P00021=-0.225,-6.128,-0.405,0.0000,0.0000,0.0000
P00022=0.222,-3.123,-1.508,0.0000,0.0000,0.0000
P00023=0.143,-0.036,0.682,0.0000,0.0000,0.0000
P00024=0.145,-0.552,1.326,0.0000,0.0000,0.0000
P00025=-2.003,0.006,0.728,0.0000,0.0000,0.0000
P00026=0.562,-0.002,-0.337,0.0000,0.0000,0.0000
P00027=-0.746,0.015,-9.096,0.0000,0.0000,0.0000
P00028=-2.237,-0.018,-7.702,0.0000,0.0000,0.0000
P00029=-2.156,-0.086,-4.681,0.0000,0.0000,0.0000
P00030=5.926,-4.294,-1.390,0.0000,0.0000,0.0000
P00031=1.853,-0.001,-1.549,0.0000,0.0000,0.0000
P00032=1.957,0.503,-7.217,0.0000,0.0000,0.0000
///RCONF 0,0,0,0,1,0,0,0,0,0,0,0,0,0,0,0,0,0,0,0,0,0,0,0
P00033=-0.123,0.612,-5.012,0.0000,0.0000,0.0000
///RCONF 0,0,0,0,0,0,0,0,0,0,0,0,0,0,0,0,0,0,0,0,0,0,0,0
P00034=-0.304,0.773,-2.693,0.0000,0.0000,0.0000
P00035=2.817,0.591,-1.622,0.0000,0.0000,0.0000
P00040=-0.030,9.648,2.467,0.0000,0.0000,0.0000
P00041=0.192,3.924,0.305,0.0000,0.0000,0.0000
P00042=-0.217,1.941,0.413,0.0000,0.0000,0.0000
P00043=-0.044,-1.937,1.197,0.0000,0.0000,0.0000
P00044=0.687,-2.322,1.156,0.0000,0.0000,0.0000
P00045=-0.068,-0.810,1.603,0.0000,0.0000,0.0000
P00046=0.799,0.043,1.292,0.0000,0.0000,0.0000
///RCONF 0,1,0,0,0,0,0,0,0,0,0,0,0,0,0,0,0,0,0,0,0,0,0,0
P00047=-0.011,1.737,-0.646,0.0000,0.0000,0.0000
///RCONF 0,0,0,0,0,0,0,0,0,0,0,0,0,0,0,0,0,0,0,0,0,0,0,0
P00048=2.411,0.025,-0.606,0.0000,0.0000,0.0000
P00049=3.413,-3.572,-1.618,0.0000,0.0000,0.0000
P00050=4.296,-4.501,-0.826,0.0000,0.0000,0.0000
P00051=0.367,3.892,0.009,0.0000,0.0000,0.0000
P00052=0.088,2.832,-0.342,0.0000,0.0000,0.0000
P00053=0.134,6.594,0.107,0.0000,0.0000,0.0000
P00054=-0.103,6.509,-0.702,0.0000,0.0000,0.0000
P00061=1.575,-3.405,-0.752,0.0000,0.0000,0.0000
P00062=-0.135,-0.848,-1.706,0.0000,0.0000,0.0000
P00063=0.036,-0.654,-3.005,0.0000,0.0000,0.0000
P00069=2.004,-0.013,0.498,0.0000,0.0000,0.0000
P00071=2.716,0.070,1.352,0.0000,0.0000,0.0000
P00072=1.041,-0.003,-0.797,0.0000,0.0000,0.0000
P00073=-0.961,5.319,-6.157,0.0000,0.0000,0.0000
P00074=1.123,1.944,-5.914,0.0000,0.0000,0.0000
P00080=-3.893,-3.240,-0.208,0.0000,0.0000,0.0000
P00081=19.486,11.347,1.262,0.0000,0.0000,0.0000
P00095=-3.945,4.918,-0.177,0.0000,0.0000,0.0000
P00096=-0.633,5.398,-3.809,0.0000,0.0000,0.0000
//INST
///DATE 2024/08/30 08:22
///ATTR SC,RW
///GROUP1 RB1,BS1
///GROUP2 ST1
NOP
'X2_8A-21A(90,0)
MOVJ C00000 BC00000 VJ=100.00  +MOVJ EC00000 VJ=100.00
CALL JOB:CLEAN-R1_KM_NEW
MOVJ C00001 BC00001 VJ=100.00  +MOVJ EC00001 VJ=100.00
MOVJ C00002 BC00002 VJ=100.00  +MOVJ EC00002 VJ=100.00
'Path S3463
SFTOF3D
MOVJ C00003 BC00003 VJ=100.00  +MOVJ EC00003 VJ=100.00
MOVL C00004 BC00004 V=666.7  +MOVJ EC00004 VJ=100.00
SMOVL C00005 BC00005 V=166.7  +MOVJ EC00005
SREFP 3 C00006 BC00006  +REFP EC00006
CALL JOB:SEARCH-R1-S13D
SET P095 P006
SFTON3D P095
SMOVL C00007 BC00007 V=166.7  +MOVJ EC00007
SMOVL C00008 BC00008 V=166.7  +MOVJ EC00008
SREFP 3 C00009 BC00009  +REFP EC00009
CALL JOB:SEARCH-R1-S13D
SET P095 P006
SFTON3D P095
SMOVL C00010 BC00010 V=166.7  +MOVJ EC00010
MOVL C00011 BC00011 V=1000.0  +MOVJ EC00011 VJ=100.00
'EndPath S3463
'Path S3464
SFTOF3D
MOVJ C00012 BC00012 VJ=100.00  +MOVJ EC00012 VJ=100.00
MOVL C00013 BC00013 V=666.7  +MOVJ EC00013 VJ=100.00
SMOVL C00014 BC00014 V=166.7  +MOVJ EC00014
SREFP 3 C00015 BC00015  +REFP EC00015
CALL JOB:SEARCH-R1-S13D
SET P096 P006
SFTON3D P096
SMOVL C00016 BC00016 V=166.7  +MOVJ EC00016
SREFP 3 C00017 BC00017  +REFP EC00017
CALL JOB:SEARCH-R1-S13D
SET P096 P006
SFTON3D P096
SMOVL C00018 BC00018 V=166.7  +MOVJ EC00018
MOVL C00019 BC00019 V=1000.0  +MOVJ EC00019 VJ=100.00
'EndPath S3464
'Path S3465
SFTOF3D
MOVJ C00020 BC00020 VJ=100.00  +MOVJ EC00020 VJ=100.00
MOVL C00021 BC00021 V=666.7  +MOVJ EC00021 VJ=100.00
SMOVL C00022 BC00022 V=166.7  +MOVJ EC00022
SREFP 3 C00023 BC00023  +REFP EC00023
CALL JOB:SEARCH-R1-S13D
SET P021 P006
SFTON3D P021
SMOVL C00024 BC00024 V=166.7  +MOVJ EC00024
SMOVL C00025 BC00025 V=166.7  +MOVJ EC00025
SREFP 3 C00026 BC00026  +REFP EC00026
CALL JOB:SEARCH-R1-S13D
SET P021 P006
SFTON3D P021
SMOVL C00027 BC00027 V=166.7  +MOVJ EC00027
MOVL C00028 BC00028 V=1000.0  +MOVJ EC00028 VJ=100.00
'EndPath S3465
'Path S3464
SFTOF3D
MOVJ C00029 BC00029 VJ=100.00  +MOVJ EC00029 VJ=100.00
MOVL C00030 BC00030 V=666.7  +MOVJ EC00030 VJ=100.00
SMOVL C00031 BC00031 V=166.7  +MOVJ EC00031
SREFP 3 C00032 BC00032  +REFP EC00032
CALL JOB:SEARCH-R1-S13D
SET P022 P006
SFTON3D P022
SMOVL C00033 BC00033 V=166.7  +MOVJ EC00033
SREFP 3 C00034 BC00034  +REFP EC00034
CALL JOB:SEARCH-R1-S13D
SET P022 P006
SFTON3D P022
SMOVL C00035 BC00035 V=166.7  +MOVJ EC00035
MOVL C00036 BC00036 V=1000.0  +MOVJ EC00036 VJ=100.00
'EndPath S3464
MOVJ C00037 BC00037 VJ=100.00  +MOVJ EC00037 VJ=100.00
'Path S3465
SFTOF3D
MOVJ C00038 BC00038 VJ=100.00  +MOVJ EC00038 VJ=100.00
MOVL C00039 BC00039 V=666.7  +MOVJ EC00039 VJ=100.00
SMOVL C00040 BC00040 V=166.7  +MOVJ EC00040
SREFP 3 C00041 BC00041  +REFP EC00041
CALL JOB:SEARCH-R1-S13D
SET P050 P006
SFTON3D P050
SMOVL C00042 BC00042 V=166.7  +MOVJ EC00042
SREFP 3 C00043 BC00043  +REFP EC00043
CALL JOB:SEARCH-R1-S13D
SET P050 P006
SFTON3D P050
SMOVL C00044 BC00044 V=166.7  +MOVJ EC00044
SMOVL C00045 BC00045 V=166.7  +MOVJ EC00045
SREFP 3 C00046 BC00046  +REFP EC00046
CALL JOB:SEARCH-R1-S13D
SET P050 P006
SFTON3D P050
SMOVL C00047 BC00047 V=166.7  +MOVJ EC00047
MOVL C00048 BC00048 V=1000.0  +MOVJ EC00048 VJ=100.00
'EndPath S3465
'Path S3466
SFTOF3D
MOVJ C00049 BC00049 VJ=100.00  +MOVJ EC00049 VJ=100.00
MOVL C00050 BC00050 V=666.7  +MOVJ EC00050 VJ=100.00
SMOVL C00051 BC00051 V=166.7  +MOVJ EC00051
SREFP 3 C00052 BC00052  +REFP EC00052
CALL JOB:SEARCH-R1-S13D
SET P051 P006
SFTON3D P051
SMOVL C00053 BC00053 V=166.7  +MOVJ EC00053
SREFP 3 C00054 BC00054  +REFP EC00054
CALL JOB:SEARCH-R1-S13D
SET P051 P006
SFTON3D P051
SMOVL C00055 BC00055 V=166.7  +MOVJ EC00055
SMOVL C00056 BC00056 V=250.0  +MOVJ EC00056
SREFP 3 C00057 BC00057  +REFP EC00057
CALL JOB:SEARCH-R1-S13D
SET P051 P006
SFTON3D P051
SMOVL C00058 BC00058 V=166.7  +MOVJ EC00058
MOVL C00059 BC00059 V=1000.0  +MOVJ EC00059 VJ=100.00
'EndPath S3466
MOVJ C00060 BC00060 VJ=100.00  +MOVJ EC00060 VJ=100.00
MOVJ C00061 BC00061 VJ=100.00  +MOVJ EC00061 VJ=100.00
'Path S3467
SFTOF3D
MOVJ C00062 BC00062 VJ=100.00  +MOVJ EC00062 VJ=100.00
MOVL C00063 BC00063 V=666.7  +MOVJ EC00063 VJ=100.00
SMOVL C00064 BC00064 V=166.7  +MOVJ EC00064
SREFP 3 C00065 BC00065  +REFP EC00065
CALL JOB:SEARCH-R1-S13D
SET P054 P006
SFTON3D P054
SMOVL C00066 BC00066 V=250.0  +MOVJ EC00066
SMOVL C00067 BC00067 V=166.7  +MOVJ EC00067
SREFP 3 C00068 BC00068  +REFP EC00068
CALL JOB:SEARCH-R1-S13D
SET P054 P006
SFTON3D P054
SMOVL C00069 BC00069 V=166.7  +MOVJ EC00069
SMOVL C00070 BC00070 V=800.0  +MOVJ EC00070
SMOVL C00071 BC00071 V=166.7  +MOVJ EC00071
SREFP 3 C00072 BC00072  +REFP EC00072
CALL JOB:SEARCH-R1-S13D
SET P054 P006
SFTON3D P054
SMOVL C00073 BC00073 V=166.7  +MOVJ EC00073
MOVL C00074 BC00074 V=1000.0  +MOVJ EC00074 VJ=100.00
'EndPath S3467
'Path S3475
SFTOF3D
MOVJ C00075 BC00075 VJ=100.00  +MOVJ EC00075 VJ=100.00
MOVL C00076 BC00076 V=666.7  +MOVJ EC00076 VJ=100.00
SMOVL C00077 BC00077 V=166.7  +MOVJ EC00077
SREFP 3 C00078 BC00078  +REFP EC00078
CALL JOB:SEARCH-R1-S13D
SET P034 P006
SFTON3D P034
SMOVL C00079 BC00079 V=166.7  +MOVJ EC00079
SMOVL C00080 BC00080 V=333.3  +MOVJ EC00080
SMOVL C00081 BC00081 V=166.7  +MOVJ EC00081
SREFP 3 C00082 BC00082  +REFP EC00082
CALL JOB:SEARCH-R1-S13D
SET P034 P006
SFTON3D P034
SMOVL C00083 BC00083 V=166.7  +MOVJ EC00083
SMOVL C00084 BC00084 V=166.7  +MOVJ EC00084
SREFP 3 C00085 BC00085  +REFP EC00085
CALL JOB:SEARCH-R1-S13D
SET P034 P006
SFTON3D P034
SMOVL C00086 BC00086 V=166.7  +MOVJ EC00086
MOVL C00087 BC00087 V=1000.0  +MOVJ EC00087 VJ=100.00
'EndPath S3475
'Path S3464
SFTOF3D
MOVJ C00088 BC00088 VJ=100.00  +MOVJ EC00088 VJ=100.00
MOVL C00089 BC00089 V=666.7  +MOVJ EC00089 VJ=100.00
SMOVL C00090 BC00090 V=166.7  +MOVJ EC00090
SREFP 3 C00091 BC00091  +REFP EC00091
CALL JOB:SEARCH-R1-S13D
SET P023 P006
SFTON3D P023
SMOVL C00092 BC00092 V=166.7  +MOVJ EC00092
SMOVL C00093 BC00093 V=500.0  +MOVJ EC00093
SMOVL C00094 BC00094 V=166.7  +MOVJ EC00094
SREFP 3 C00095 BC00095  +REFP EC00095
CALL JOB:SEARCH-R1-S13D
SET P023 P006
SFTON3D P023
SMOVL C00096 BC00096 V=166.7  +MOVJ EC00096
SMOVL C00097 BC00097 V=166.7  +MOVJ EC00097
SREFP 3 C00098 BC00098  +REFP EC00098
CALL JOB:SEARCH-R1-S13D
SET P023 P006
SFTON3D P023
SMOVL C00099 BC00099 V=166.7  +MOVJ EC00099
MOVL C00100 BC00100 V=1000.0  +MOVJ EC00100 VJ=100.00
MOVJ C00101 BC00101 VJ=80.00  +MOVJ EC00101 VJ=80.00
MOVJ C00102 BC00102 VJ=80.00  +MOVJ EC00102 VJ=80.00
SFTOF3D
MOVJ C00103 BC00103 VJ=80.00  +MOVJ EC00103 VJ=80.00
SMOVL C00104 BC00104 V=166.7  +MOVJ EC00104
SREFP 3 C00105 BC00105  +REFP EC00105
CALL JOB:SEARCH-R1-S13D
SET P061 P006
SFTON3D P061
SMOVL C00106 BC00106 V=166.7  +MOVJ EC00106
SREFP 3 C00107 BC00107  +REFP EC00107
CALL JOB:SEARCH-R1-S13D
SET P061 P006
SFTON3D P061
SMOVL C00108 BC00108 V=166.7  +MOVJ EC00108
SFTOF3D
SMOVL C00109 BC00109 V=500.0  +MOVJ EC00109
SMOVL C00110 BC00110 V=166.7  +MOVJ EC00110
SREFP 3 C00111 BC00111  +REFP EC00111
CALL JOB:SEARCH-R1-S13D
SET P062 P006
SFTON3D P062
SMOVL C00112 BC00112 V=166.7  +MOVJ EC00112
SREFP 3 C00113 BC00113  +REFP EC00113
CALL JOB:SEARCH-R1-S13D
SET P062 P006
SFTON3D P062
SMOVL C00114 BC00114 V=166.7  +MOVJ EC00114
SFTOF3D
SMOVL C00115 BC00115 V=500.0  +MOVJ EC00115
SMOVL C00116 BC00116 V=166.7  +MOVJ EC00116
SREFP 3 C00117 BC00117  +REFP EC00117
CALL JOB:SEARCH-R1-S13D
SET P063 P006
SFTON3D P063
SMOVL C00118 BC00118 V=166.7  +MOVJ EC00118
SREFP 3 C00119 BC00119  +REFP EC00119
CALL JOB:SEARCH-R1-S13D
SET P063 P006
SFTON3D P063
SMOVL C00120 BC00120 V=166.7  +MOVJ EC00120
SFTOF3D
SMOVL C00121 BC00121 V=500.0  +MOVJ EC00121
MOVJ C00122 BC00122 VJ=80.00  +MOVJ EC00122 VJ=80.00
MOVJ C00123 BC00123 VJ=80.00  +MOVJ EC00123 VJ=80.00
'EndPath S3464
MOVJ C00124 BC00124 VJ=100.00  +MOVJ EC00124 VJ=100.00
'Path S3465
SFTOF3D
MOVJ C00125 BC00125 VJ=100.00  +MOVJ EC00125 VJ=100.00
MOVL C00126 BC00126 V=666.7  +MOVJ EC00126 VJ=100.00
SMOVL C00127 BC00127 V=166.7  +MOVJ EC00127
SREFP 3 C00128 BC00128  +REFP EC00128
CALL JOB:SEARCH-R1-S13D
SET P024 P006
SFTON3D P024
SMOVL C00129 BC00129 V=166.7  +MOVJ EC00129
SREFP 3 C00130 BC00130  +REFP EC00130
CALL JOB:SEARCH-R1-S13D
SET P024 P006
SFTON3D P024
SMOVL C00131 BC00131 V=166.7  +MOVJ EC00131
SMOVL C00132 BC00132 V=166.7  +MOVJ EC00132
SREFP 3 C00133 BC00133  +REFP EC00133
CALL JOB:SEARCH-R1-S13D
SET P024 P006
SFTON3D P024
SMOVL C00134 BC00134 V=166.7  +MOVJ EC00134
MOVL C00135 BC00135 V=1000.0  +MOVJ EC00135 VJ=100.00
'EndPath S3465
'Path S3476
SFTOF3D
MOVJ C00136 BC00136 VJ=100.00  +MOVJ EC00136 VJ=100.00
MOVL C00137 BC00137 V=666.7  +MOVJ EC00137 VJ=100.00
SMOVL C00138 BC00138 V=166.7  +MOVJ EC00138
SREFP 3 C00139 BC00139  +REFP EC00139
CALL JOB:SEARCH-R1-S13D
SET P035 P006
SFTON3D P035
SMOVL C00140 BC00140 V=166.7  +MOVJ EC00140
SREFP 3 C00141 BC00141  +REFP EC00141
CALL JOB:SEARCH-R1-S13D
SET P035 P006
SFTON3D P035
SMOVL C00142 BC00142 V=166.7  +MOVJ EC00142
SMOVL C00143 BC00143 V=333.3  +MOVJ EC00143
SMOVL C00144 BC00144 V=166.7  +MOVJ EC00144
SREFP 3 C00145 BC00145  +REFP EC00145
CALL JOB:SEARCH-R1-S13D
SET P035 P006
SFTON3D P035
SMOVL C00146 BC00146 V=166.7  +MOVJ EC00146
MOVL C00147 BC00147 V=1000.0  +MOVJ EC00147 VJ=100.00
'EndPath S3476
'Path S3470
SFTOF3D
MOVJ C00148 BC00148 VJ=100.00  +MOVJ EC00148 VJ=100.00
MOVL C00149 BC00149 V=666.7  +MOVJ EC00149 VJ=100.00
SMOVL C00150 BC00150 V=166.7  +MOVJ EC00150
SREFP 3 C00151 BC00151  +REFP EC00151
CALL JOB:SEARCH-R1-S13D
SET P029 P006
SFTON3D P029
SMOVL C00152 BC00152 V=166.7  +MOVJ EC00152
SREFP 3 C00153 BC00153  +REFP EC00153
CALL JOB:SEARCH-R1-S13D
SET P029 P006
SFTON3D P029
SMOVL C00154 BC00154 V=166.7  +MOVJ EC00154
SMOVL C00155 BC00155 V=250.0  +MOVJ EC00155
SMOVL C00156 BC00156 V=166.7  +MOVJ EC00156
SREFP 3 C00157 BC00157  +REFP EC00157
CALL JOB:SEARCH-R1-S13D
SET P029 P006
SFTON3D P029
SMOVL C00158 BC00158 V=166.7  +MOVJ EC00158
MOVL C00159 BC00159 V=1000.0  +MOVJ EC00159 VJ=100.00
'EndPath S3470
'Path S4850
SFTOF3D
MOVL C00160 BC00160 V=666.7  +MOVJ EC00160 VJ=100.00
SMOVL C00161 BC00161 V=166.7  +MOVJ EC00161
SREFP 3 C00162 BC00162  +REFP EC00162
CALL JOB:SEARCH-R1-S13D
SET P071 P006
SFTON3D P071
SMOVL C00163 BC00163 V=166.7  +MOVJ EC00163
SREFP 3 C00164 BC00164  +REFP EC00164
CALL JOB:SEARCH-R1-S13D
SET P071 P006
SFTON3D P071
SMOVL C00165 BC00165 V=166.7  +MOVJ EC00165
SMOVL C00166 BC00166 V=166.7  +MOVJ EC00166
SREFP 3 C00167 BC00167  +REFP EC00167
CALL JOB:SEARCH-R1-S13D
SET P071 P006
SFTON3D P071
SMOVL C00168 BC00168 V=166.7  +MOVJ EC00168
MOVL C00169 BC00169 V=1000.0  +MOVJ EC00169 VJ=100.00
'EndPath S4850
'Path S4851
SFTOF3D
MOVJ C00170 BC00170 VJ=100.00  +MOVJ EC00170 VJ=100.00
'POMIAR_DOD_WZM_BOK
MOVL C00171 BC00171 V=666.7  +MOVJ EC00171 VJ=100.00
SMOVL C00172 BC00172 V=166.7  +MOVJ EC00172
SREFP 3 C00173 BC00173  +REFP EC00173
CALL JOB:SEARCH-R1-S13D
SET P080 P006
SFTON3D P080
SMOVL C00174 BC00174 V=166.7  +MOVJ EC00174
SREFP 3 C00175 BC00175  +REFP EC00175
CALL JOB:SEARCH-R1-S13D
SET P080 P006
SFTON3D P080
SMOVL C00176 BC00176 V=166.7  +MOVJ EC00176
SMOVL C00177 BC00177 V=250.0  +MOVJ EC00177
SMOVL C00178 BC00178 V=166.7  +MOVJ EC00178
SREFP 3 C00179 BC00179  +REFP EC00179
CALL JOB:SEARCH-R1-S13D
SET P080 P006
SFTON3D P080
SMOVL C00180 BC00180 V=166.7  +MOVJ EC00180
MOVL C00181 BC00181 V=1000.0  +MOVJ EC00181 VJ=100.00
SFTOF3D
MOVJ C00182 BC00182 VJ=100.00  +MOVJ EC00182 VJ=100.00
MOVL C00183 BC00183 V=666.7  +MOVJ EC00183 VJ=100.00
SMOVL C00184 BC00184 V=166.7  +MOVJ EC00184
SREFP 3 C00185 BC00185  +REFP EC00185
CALL JOB:SEARCH-R1-S13D
SET P072 P006
SFTON3D P072
SMOVL C00186 BC00186 V=166.7  +MOVJ EC00186
SREFP 3 C00187 BC00187  +REFP EC00187
CALL JOB:SEARCH-R1-S13D
SET P072 P006
SFTON3D P072
SMOVL C00188 BC00188 V=166.7  +MOVJ EC00188
MOVL C00189 BC00189 V=1000.0  +MOVJ EC00189 VJ=100.00
'EndPath S4851
MOVJ C00190 BC00190 VJ=100.00  +MOVJ EC00190 VJ=100.00
MOVJ C00191 BC00191 VJ=100.00  +MOVJ EC00191 VJ=100.00
'Path S4852
SFTOF3D
MOVJ C00192 BC00192 VJ=100.00  +MOVJ EC00192 VJ=100.00
MOVL C00193 BC00193 V=666.7  +MOVJ EC00193 VJ=100.00
SMOVL C00194 BC00194 V=166.7  +MOVJ EC00194
SREFP 3 C00195 BC00195  +REFP EC00195
CALL JOB:SEARCH-R1-S13D
SET P073 P006
SFTON3D P073
SMOVL C00196 BC00196 V=166.7  +MOVJ EC00196
SMOVL C00197 BC00197 V=166.7  +MOVJ EC00197
SREFP 3 C00198 BC00198  +REFP EC00198
CALL JOB:SEARCH-R1-S13D
SET P073 P006
SFTON3D P073
SMOVL C00199 BC00199 V=166.7  +MOVJ EC00199
SMOVL C00200 BC00200 V=166.7  +MOVJ EC00200
SREFP 3 C00201 BC00201  +REFP EC00201
CALL JOB:SEARCH-R1-S13D
SET P073 P006
SFTON3D P073
SMOVL C00202 BC00202 V=166.7  +MOVJ EC00202
MOVL C00203 BC00203 V=1000.0  +MOVJ EC00203 VJ=100.00
'EndPath S4852
MOVJ C00204 BC00204 VJ=100.00  +MOVJ EC00204 VJ=100.00
'Path S4853
SFTOF3D
MOVJ C00205 BC00205 VJ=100.00  +MOVJ EC00205 VJ=100.00
MOVL C00206 BC00206 V=666.7  +MOVJ EC00206 VJ=100.00
SMOVL C00207 BC00207 V=166.7  +MOVJ EC00207
SREFP 3 C00208 BC00208  +REFP EC00208
CALL JOB:SEARCH-R1-S13D
SET P074 P006
SFTON3D P074
SMOVL C00209 BC00209 V=166.7  +MOVJ EC00209
SREFP 3 C00210 BC00210  +REFP EC00210
CALL JOB:SEARCH-R1-S13D
SET P074 P006
SFTON3D P074
SMOVL C00211 BC00211 V=166.7  +MOVJ EC00211
MOVL C00212 BC00212 V=1000.0  +MOVJ EC00212 VJ=100.00
'EndPath S4853
'Path S3467
SFTOF3D
MOVJ C00213 BC00213 VJ=100.00  +MOVJ EC00213 VJ=100.00
MOVJ C00214 BC00214 VJ=100.00  +MOVJ EC00214 VJ=100.00
MOVL C00215 BC00215 V=666.7  +MOVJ EC00215 VJ=100.00
SMOVL C00216 BC00216 V=166.7  +MOVJ EC00216
SREFP 3 C00217 BC00217  +REFP EC00217
CALL JOB:SEARCH-R1-S13D
SET P081 P006
SFTON3D P081
SMOVL C00218 BC00218 V=166.7  +MOVJ EC00218
SMOVL C00219 BC00219 V=166.7  +MOVJ EC00219
SREFP 3 C00220 BC00220  +REFP EC00220
CALL JOB:SEARCH-R1-S13D
SET P081 P006
SFTON3D P081
SMOVL C00221 BC00221 V=166.7  +MOVJ EC00221
SMOVL C00222 BC00222 V=800.0  +MOVJ EC00222
SMOVL C00223 BC00223 V=166.7  +MOVJ EC00223
SREFP 3 C00224 BC00224  +REFP EC00224
CALL JOB:SEARCH-R1-S13D
SET P081 P006
SFTON3D P081
SMOVL C00225 BC00225 V=166.7  +MOVJ EC00225
MOVJ C00226 BC00226 VJ=100.00  +MOVJ EC00226 VJ=100.00
MOVJ C00227 BC00227 VJ=100.00  +MOVJ EC00227 VJ=100.00
SFTOF3D
MOVJ C00228 BC00228 VJ=100.00  +MOVJ EC00228 VJ=100.00
MOVL C00229 BC00229 V=666.7  +MOVJ EC00229 VJ=100.00
SMOVL C00230 BC00230 V=166.7  +MOVJ EC00230
SREFP 3 C00231 BC00231  +REFP EC00231
CALL JOB:SEARCH-R1-S13D
SET P026 P006
SFTON3D P026
SMOVL C00232 BC00232 V=166.7  +MOVJ EC00232
SREFP 3 C00233 BC00233  +REFP EC00233
CALL JOB:SEARCH-R1-S13D
SET P026 P006
SFTON3D P026
SMOVL C00234 BC00234 V=166.7  +MOVJ EC00234
SMOVL C00235 BC00235 V=800.0  +MOVJ EC00235
SMOVL C00236 BC00236 V=166.7  +MOVJ EC00236
SREFP 3 C00237 BC00237  +REFP EC00237
CALL JOB:SEARCH-R1-S13D
SET P026 P006
SFTON3D P026
SMOVL C00238 BC00238 V=166.7  +MOVJ EC00238
MOVL C00239 BC00239 V=1000.0  +MOVJ EC00239 VJ=100.00
'EndPath S3467
MOVJ C00240 BC00240 VJ=100.00  +MOVJ EC00240 VJ=100.00
'Path S3466
SFTOF3D
MOVJ C00241 BC00241 VJ=100.00  +MOVJ EC00241 VJ=100.00
MOVL C00242 BC00242 V=666.7  +MOVJ EC00242 VJ=100.00
SMOVL C00243 BC00243 V=166.7  +MOVJ EC00243
SREFP 3 C00244 BC00244  +REFP EC00244
CALL JOB:SEARCH-R1-S13D
SET P025 P006
SFTON3D P025
SMOVL C00245 BC00245 V=166.7  +MOVJ EC00245
SMOVL C00246 BC00246 V=166.7  +MOVJ EC00246
SREFP 3 C00247 BC00247  +REFP EC00247
CALL JOB:SEARCH-R1-S13D
SET P025 P006
SFTON3D P025
SMOVL C00248 BC00248 V=166.7  +MOVJ EC00248
SMOVL C00249 BC00249 V=200.0  +MOVJ EC00249
SMOVL C00250 BC00250 V=166.7  +MOVJ EC00250
SREFP 3 C00251 BC00251  +REFP EC00251
CALL JOB:SEARCH-R1-S13D
SET P025 P006
SFTON3D P025
SMOVL C00252 BC00252 V=166.7  +MOVJ EC00252
MOVL C00253 BC00253 V=1000.0  +MOVJ EC00253 VJ=100.00
'EndPath S3466
MOVJ C00254 BC00254 VJ=100.00  +MOVJ EC00254 VJ=100.00
'Path S3469
SFTOF3D
MOVJ C00255 BC00255 VJ=100.00  +MOVJ EC00255 VJ=100.00
MOVL C00256 BC00256 V=666.7  +MOVJ EC00256 VJ=100.00
SMOVL C00257 BC00257 V=166.7  +MOVJ EC00257
SREFP 3 C00258 BC00258  +REFP EC00258
CALL JOB:SEARCH-R1-S13D
SET P028 P006
SFTON3D P028
SMOVL C00259 BC00259 V=166.7  +MOVJ EC00259
SREFP 3 C00260 BC00260  +REFP EC00260
CALL JOB:SEARCH-R1-S13D
SET P028 P006
SFTON3D P028
SMOVL C00261 BC00261 V=166.7  +MOVJ EC00261
SMOVL C00262 BC00262 V=333.3  +MOVJ EC00262
SMOVL C00263 BC00263 V=166.7  +MOVJ EC00263
SREFP 3 C00264 BC00264  +REFP EC00264
CALL JOB:SEARCH-R1-S13D
SET P028 P006
SFTON3D P028
SMOVL C00265 BC00265 V=166.7  +MOVJ EC00265
MOVL C00266 BC00266 V=1000.0  +MOVJ EC00266 VJ=100.00
'EndPath S3469
MOVJ C00267 BC00267 VJ=100.00  +MOVJ EC00267 VJ=100.00
'Path S3474
SFTOF3D
MOVJ C00268 BC00268 VJ=100.00  +MOVJ EC00268 VJ=100.00
MOVL C00269 BC00269 V=666.7  +MOVJ EC00269 VJ=100.00
SMOVL C00270 BC00270 V=166.7  +MOVJ EC00270
SREFP 3 C00271 BC00271  +REFP EC00271
CALL JOB:SEARCH-R1-S13D
SET P033 P006
SFTON3D P033
SMOVL C00272 BC00272 V=166.7  +MOVJ EC00272
SREFP 3 C00273 BC00273  +REFP EC00273
CALL JOB:SEARCH-R1-S13D
SET P033 P006
SFTON3D P033
SMOVL C00274 BC00274 V=166.7  +MOVJ EC00274
SMOVL C00275 BC00275 V=250.0  +MOVJ EC00275
SMOVL C00276 BC00276 V=166.7  +MOVJ EC00276
SREFP 3 C00277 BC00277  +REFP EC00277
CALL JOB:SEARCH-R1-S13D
SET P033 P006
SFTON3D P033
SMOVL C00278 BC00278 V=166.7  +MOVJ EC00278
MOVL C00279 BC00279 V=1000.0  +MOVJ EC00279 VJ=100.00
'EndPath S3474
'Path S3468
SFTOF3D
MOVJ C00280 BC00280 VJ=100.00  +MOVJ EC00280 VJ=100.00
MOVL C00281 BC00281 V=666.7  +MOVJ EC00281 VJ=100.00
SMOVL C00282 BC00282 V=166.7  +MOVJ EC00282
SREFP 3 C00283 BC00283  +REFP EC00283
CALL JOB:SEARCH-R1-S13D
SET P027 P006
SFTON3D P027
SMOVL C00284 BC00284 V=166.7  +MOVJ EC00284
SMOVL C00285 BC00285 V=166.7  +MOVJ EC00285
SREFP 3 C00286 BC00286  +REFP EC00286
CALL JOB:SEARCH-R1-S13D
SET P027 P006
SFTON3D P027
SMOVL C00287 BC00287 V=166.7  +MOVJ EC00287
SMOVL C00288 BC00288 V=166.7  +MOVJ EC00288
SREFP 3 C00289 BC00289  +REFP EC00289
CALL JOB:SEARCH-R1-S13D
SET P027 P006
SFTON3D P027
SMOVL C00290 BC00290 V=166.7  +MOVJ EC00290
MOVL C00291 BC00291 V=1000.0  +MOVJ EC00291 VJ=100.00
'EndPath S3468
'Path S3471
SFTOF3D
MOVJ C00292 BC00292 VJ=100.00  +MOVJ EC00292 VJ=100.00
MOVL C00293 BC00293 V=666.7  +MOVJ EC00293 VJ=100.00
SMOVL C00294 BC00294 V=166.7  +MOVJ EC00294
SREFP 3 C00295 BC00295  +REFP EC00295
CALL JOB:SEARCH-R1-S13D
SET P030 P006
SFTON3D P030
SMOVL C00296 BC00296 V=166.7  +MOVJ EC00296
SREFP 3 C00297 BC00297  +REFP EC00297
CALL JOB:SEARCH-R1-S13D
SET P030 P006
SFTON3D P030
SMOVL C00298 BC00298 V=166.7  +MOVJ EC00298
MOVL C00299 BC00299 V=1000.0  +MOVJ EC00299 VJ=100.00
'EndPath S3471
'Path S3472
SFTOF3D
MOVJ C00300 BC00300 VJ=100.00  +MOVJ EC00300 VJ=100.00
MOVL C00301 BC00301 V=666.7  +MOVJ EC00301 VJ=100.00
SMOVL C00302 BC00302 V=166.7  +MOVJ EC00302
SREFP 3 C00303 BC00303  +REFP EC00303
CALL JOB:SEARCH-R1-S13D
SET P031 P006
SFTON3D P031
SMOVL C00304 BC00304 V=166.7  +MOVJ EC00304
SREFP 3 C00305 BC00305  +REFP EC00305
CALL JOB:SEARCH-R1-S13D
SET P031 P006
SFTON3D P031
SMOVL C00306 BC00306 V=166.7  +MOVJ EC00306
MOVL C00307 BC00307 V=1000.0  +MOVJ EC00307 VJ=100.00
'EndPath S3472
MOVJ C00308 BC00308 VJ=100.00  +MOVJ EC00308 VJ=100.00
'Path S3472
SFTOF3D
MOVJ C00309 BC00309 VJ=100.00  +MOVJ EC00309 VJ=100.00
MOVL C00310 BC00310 V=666.7  +MOVJ EC00310 VJ=100.00
SMOVL C00311 BC00311 V=166.7  +MOVJ EC00311
SREFP 3 C00312 BC00312  +REFP EC00312
CALL JOB:SEARCH-R1-S13D
SET P032 P006
SFTON3D P032
SMOVL C00313 BC00313 V=166.7  +MOVJ EC00313
SREFP 3 C00314 BC00314  +REFP EC00314
CALL JOB:SEARCH-R1-S13D
SET P032 P006
SFTON3D P032
SMOVL C00315 BC00315 V=166.7  +MOVJ EC00315
SMOVL C00316 BC00316 V=133.3  +MOVJ EC00316
SREFP 3 C00317 BC00317  +REFP EC00317
CALL JOB:SEARCH-R1-S13D
SET P032 P006
SFTON3D P032
SMOVL C00318 BC00318 V=166.7  +MOVJ EC00318
MOVL C00319 BC00319 V=1000.0  +MOVJ EC00319 VJ=100.00
'EndPath S3472
MOVJ C00320 BC00320 VJ=100.00  +MOVJ EC00320 VJ=100.00
'Path S3477
SFTOF3D
MOVJ C00321 BC00321 VJ=100.00  +MOVJ EC00321 VJ=100.00
SMOVL C00322 BC00322 V=166.7  +MOVJ EC00322
SREFP 3 C00323 BC00323  +REFP EC00323
CALL JOB:SEARCH-R1-S13D
SET P069 P006
SFTON3D P069
SMOVL C00324 BC00324 V=250.0  +MOVJ EC00324
SMOVL C00325 BC00325 V=250.0  +MOVJ EC00325
SMOVL C00326 BC00326 V=166.7  +MOVJ EC00326
SREFP 3 C00327 BC00327  +REFP EC00327
CALL JOB:SEARCH-R1-S13D
SET P069 P006
SFTON3D P069
SMOVL C00328 BC00328 V=166.7  +MOVJ EC00328
SFTOF3D
SMOVL C00329 BC00329 V=666.7  +MOVJ EC00329
MOVL C00330 BC00330 V=666.7  +MOVJ EC00330 VJ=100.00
SMOVL C00331 BC00331 V=166.7  +MOVJ EC00331
SREFP 3 C00332 BC00332  +REFP EC00332
CALL JOB:SEARCH-R1-S13D
SET P052 P006
SFTON3D P052
SMOVL C00333 BC00333 V=166.7  +MOVJ EC00333
SREFP 3 C00334 BC00334  +REFP EC00334
CALL JOB:SEARCH-R1-S13D
SET P052 P006
SFTON3D P052
SMOVL C00335 BC00335 V=166.7  +MOVJ EC00335
MOVL C00336 BC00336 V=1000.0  +MOVJ EC00336 VJ=100.00
'EndPath S3477
MOVJ C00337 BC00337 VJ=100.00  +MOVJ EC00337 VJ=100.00
'poprawiÄ searcha- nie mialem
'wyciecia
'Path S3478
SFTOF3D
MOVJ C00338 BC00338 VJ=100.00  +MOVJ EC00338 VJ=100.00
MOVL C00339 BC00339 V=666.7  +MOVJ EC00339 VJ=100.00
SMOVL C00340 BC00340 V=166.7  +MOVJ EC00340
SREFP 3 C00341 BC00341  +REFP EC00341
CALL JOB:SEARCH-R1-S13D
SET P053 P006
SFTON3D P053
SMOVL C00342 BC00342 V=166.7  +MOVJ EC00342
SREFP 3 C00343 BC00343  +REFP EC00343
CALL JOB:SEARCH-R1-S13D
SET P053 P006
SFTON3D P053
SMOVL C00344 BC00344 V=166.7  +MOVJ EC00344
MOVL C00345 BC00345 V=1000.0  +MOVJ EC00345 VJ=100.00
'EndPath S3478
'
MOVJ C00346 BC00346 VJ=100.00  +MOVJ EC00346 VJ=100.00
'Path W3476
SFTOF3D
SFTON3D P033
MOVJ C00347 BC00347 VJ=100.00  +MOVJ EC00347 VJ=100.00
SMOVL C00348 BC00348 V=800.0  +MOVJ EC00348
SMOVL C00349 BC00349 V=166.7 PL=0  +MOVJ EC00349
MACRO1 MJ#(0) ARGF14
ARCON
SMOVL C00350 BC00350 V=10.0  +MOVJ EC00350
ARCOF
SMOVL C00351 BC00351 V=800.0  +MOVJ EC00351
SMOVL C00352 BC00352 V=1000.0  +MOVJ EC00352
SFTOF3D
'EndPath W3476
'Path W3477
SFTOF3D
SFTON3D P033
MOVJ C00353 BC00353 VJ=100.00  +MOVJ EC00353 VJ=100.00
SMOVL C00354 BC00354 V=800.0  +MOVJ EC00354
SMOVL C00355 BC00355 V=166.7 PL=0  +MOVJ EC00355
SMOVL C00356 BC00356 V=10.0  +MOVJ EC00356
SMOVL C00357 BC00357 V=10.0  +MOVJ EC00357
SMOVL C00358 BC00358 V=10.0  +MOVJ EC00358
ARCOF
SMOVL C00359 BC00359 V=800.0  +MOVJ EC00359
SMOVL C00360 BC00360 V=1000.0  +MOVJ EC00360
SFTOF3D
'EndPath W3477
MOVJ C00361 BC00361 VJ=100.00  +MOVJ EC00361 VJ=100.00
'Path W3478
SFTOF3D
SFTON3D P033
MOVJ C00362 BC00362 VJ=100.00  +MOVJ EC00362 VJ=100.00
SMOVL C00363 BC00363 V=800.0  +MOVJ EC00363
SMOVL C00364 BC00364 V=166.7 PL=0  +MOVJ EC00364
ARCON
SMOVL C00365 BC00365 V=10.0  +MOVJ EC00365
SMOVL C00366 BC00366 V=10.0  +MOVJ EC00366
SMOVL C00367 BC00367 V=10.0  +MOVJ EC00367
ARCOF
SMOVL C00368 BC00368 V=800.0  +MOVJ EC00368
SMOVL C00369 BC00369 V=1000.0  +MOVJ EC00369
SFTOF3D
'EndPath W3478
MOVJ C00370 BC00370 VJ=100.00  +MOVJ EC00370 VJ=100.00
MOVJ C00371 BC00371 VJ=100.00  +MOVJ EC00371 VJ=100.00
SFTOF3D
SFTON3D P081
MOVJ C00372 BC00372 VJ=100.00  +MOVJ EC00372 VJ=100.00
SMOVL C00373 BC00373 V=800.0  +MOVJ EC00373
SMOVL C00374 BC00374 V=166.7 PL=0  +MOVJ EC00374
ARCON
SMOVL C00375 BC00375 V=9.2  +MOVJ EC00375
ARCOF
SMOVL C00376 BC00376 V=800.0  +MOVJ EC00376
SMOVL C00377 BC00377 V=1000.0  +MOVJ EC00377
SFTOF3D
'EndPath W3479
'Path W3480
SFTOF3D
SFTON3D P081
MOVJ C00378 BC00378 VJ=100.00  +MOVJ EC00378 VJ=100.00
SMOVL C00379 BC00379 V=800.0  +MOVJ EC00379
SMOVL C00380 BC00380 V=150.0 PL=0  +MOVJ EC00380
ARCON
SMOVL C00381 BC00381 V=10.0  +MOVJ EC00381
ARCOF
SMOVL C00382 BC00382 V=800.0  +MOVJ EC00382
SMOVL C00383 BC00383 V=1000.0  +MOVJ EC00383
SFTOF3D
'EndPath W3480
'Path W3481
SFTOF3D
SFTON3D P081
MOVJ C00384 BC00384 VJ=100.00  +MOVJ EC00384 VJ=100.00
SMOVL C00385 BC00385 V=800.0  +MOVJ EC00385
SMOVL C00386 BC00386 V=150.0 PL=0  +MOVJ EC00386
ARCON
SMOVL C00387 BC00387 V=10.0  +MOVJ EC00387
ARCOF
SMOVL C00388 BC00388 V=800.0  +MOVJ EC00388
SMOVL C00389 BC00389 V=1000.0  +MOVJ EC00389
SFTOF3D
'EndPath W3481
MOVJ C00390 BC00390 VJ=100.00  +MOVJ EC00390 VJ=100.00
'uwaga na podajnik
'Path W3481
SFTOF3D
SFTON3D P081
MOVJ C00391 BC00391 VJ=50.00  +MOVJ EC00391 VJ=15.00
SMOVL C00392 BC00392 V=800.0  +MOVJ EC00392
SMOVL C00393 BC00393 V=150.0 PL=0  +MOVJ EC00393
ARCON
SMOVL C00394 BC00394 V=10.0  +MOVJ EC00394
ARCOF
SMOVL C00395 BC00395 V=800.0  +MOVJ EC00395
SMOVL C00396 BC00396 V=1000.0  +MOVJ EC00396
SFTOF3D
'9
'Path W3479
MOVJ C00397 BC00397 VJ=100.00  +MOVJ EC00397 VJ=100.00
SFTOF3D
SFTON3D P026
MOVJ C00398 BC00398 VJ=100.00  +MOVJ EC00398 VJ=100.00
SMOVL C00399 BC00399 V=800.0  +MOVJ EC00399
SMOVL C00400 BC00400 V=166.7 PL=0  +MOVJ EC00400
ARCON
SMOVL C00401 BC00401 V=9.2  +MOVJ EC00401
SMOVL C00402 BC00402 V=9.2  +MOVJ EC00402
SMOVL C00403 BC00403 V=9.2  +MOVJ EC00403
ARCOF
SMOVL C00404 BC00404 V=800.0  +MOVJ EC00404
SMOVL C00405 BC00405 V=1000.0  +MOVJ EC00405
SFTOF3D
'EndPath W3479
'Path W3480
SFTOF3D
SFTON3D P026
MOVJ C00406 BC00406 VJ=100.00  +MOVJ EC00406 VJ=100.00
SMOVL C00407 BC00407 V=800.0  +MOVJ EC00407
SMOVL C00408 BC00408 V=150.0 PL=0  +MOVJ EC00408
ARCON
SMOVL C00409 BC00409 V=10.0  +MOVJ EC00409
SMOVL C00410 BC00410 V=10.0  +MOVJ EC00410
SMOVL C00411 BC00411 V=10.0  +MOVJ EC00411
ARCOF
SMOVL C00412 BC00412 V=800.0  +MOVJ EC00412
SMOVL C00413 BC00413 V=1000.0  +MOVJ EC00413
SFTOF3D
'EndPath W3480
'Path W3481
SFTOF3D
SFTON3D P026
MOVJ C00414 BC00414 VJ=100.00  +MOVJ EC00414 VJ=100.00
SMOVL C00415 BC00415 V=800.0  +MOVJ EC00415
SMOVL C00416 BC00416 V=150.0 PL=0  +MOVJ EC00416
ARCON
SMOVL C00417 BC00417 V=10.0  +MOVJ EC00417
ARCOF
SMOVL C00418 BC00418 V=800.0  +MOVJ EC00418
SMOVL C00419 BC00419 V=1000.0  +MOVJ EC00419
SFTOF3D
'EndPath W3481
MOVJ C00420 BC00420 VJ=100.00  +MOVJ EC00420 VJ=100.00
'uwaga na podajnik
'Path W3481
SFTOF3D
SFTON3D P026
MOVJ C00421 BC00421 VJ=50.00  +MOVJ EC00421 VJ=15.00
SMOVL C00422 BC00422 V=800.0  +MOVJ EC00422
SMOVL C00423 BC00423 V=150.0 PL=0  +MOVJ EC00423
ARCON
SMOVL C00424 BC00424 V=10.0  +MOVJ EC00424
SMOVL C00425 BC00425 V=10.0  +MOVJ EC00425
ARCOF
SMOVL C00426 BC00426 V=800.0  +MOVJ EC00426
SMOVL C00427 BC00427 V=1000.0  +MOVJ EC00427
SFTOF3D
'EndPath W3481
'brak dostepu offset drutu 1cm
'Path W3482
SFTOF3D
SFTON3D P026
MOVJ C00428 BC00428 VJ=100.00  +MOVJ EC00428 VJ=100.00
SMOVL C00429 BC00429 V=800.0  +MOVJ EC00429
SMOVL C00430 BC00430 V=150.0 PL=0  +MOVJ EC00430
ARCON
SMOVL C00431 BC00431 V=10.0  +MOVJ EC00431
ARCOF
SMOVL C00432 BC00432 V=800.0  +MOVJ EC00432
SMOVL C00433 BC00433 V=1000.0  +MOVJ EC00433
SFTOF3D
'EndPath W3482
MOVJ C00434 BC00434 VJ=100.00  +MOVJ EC00434 VJ=100.00
MOVJ C00435 BC00435 VJ=100.00  +MOVJ EC00435 VJ=100.00
'10
'11
'Path W3484
SFTOF3D
SFTON3D P025
MOVJ C00436 BC00436 VJ=100.00  +MOVJ EC00436 VJ=100.00
SMOVL C00437 BC00437 V=800.0  +MOVJ EC00437
SMOVL C00438 BC00438 V=150.0 PL=0  +MOVJ EC00438
ARCON
SMOVL C00439 BC00439 V=10.0  +MOVJ EC00439
SMOVL C00440 BC00440 V=10.0  +MOVJ EC00440
ARCOF
SMOVL C00441 BC00441 V=800.0  +MOVJ EC00441
SMOVL C00442 BC00442 V=1000.0  +MOVJ EC00442
SFTOF3D
'EndPath W3484
MOVJ C00443 BC00443 VJ=100.00  +MOVJ EC00443 VJ=100.00
'brak dostepu offset drutu 1cm
'Path W3483
SFTOF3D
SFTON3D P025
MOVJ C00444 BC00444 VJ=100.00  +MOVJ EC00444 VJ=100.00
SMOVL C00445 BC00445 V=800.0  +MOVJ EC00445
SMOVL C00446 BC00446 V=166.7 PL=0  +MOVJ EC00446
ARCON
SMOVL C00447 BC00447 V=10.0  +MOVJ EC00447
ARCOF
SMOVL C00448 BC00448 V=800.0  +MOVJ EC00448
SMOVL C00449 BC00449 V=1000.0  +MOVJ EC00449
SFTOF3D
'EndPath W3483
MOVJ C00450 BC00450 VJ=100.00  +MOVJ EC00450 VJ=100.00
MOVJ C00451 BC00451 VJ=100.00  +MOVJ EC00451 VJ=100.00
MOVJ C00452 BC00452 VJ=100.00  +MOVJ EC00452 VJ=100.00
'Path W4854
SFTOF3D
SFTON3D P073
MOVJ C00453 BC00453 VJ=100.00  +MOVJ EC00453 VJ=100.00
SMOVL C00454 BC00454 V=800.0  +MOVJ EC00454
SMOVL C00455 BC00455 V=150.0 PL=0  +MOVJ EC00455
MACRO1 MJ#(0) ARGF9
ARCON
SMOVL C00456 BC00456 V=9.2  +MOVJ EC00456
SFTON3D P074
SMOVL C00457 BC00457 V=9.2  +MOVJ EC00457
SMOVL C00458 BC00458 V=9.2  +MOVJ EC00458
ARCOF
SMOVL C00459 BC00459 V=800.0  +MOVJ EC00459
MOVJ C00460 BC00460 VJ=50.00  +MOVJ EC00460 VJ=100.00
SMOVL C00461 BC00461 V=166.7  +MOVJ EC00461
SMOVL C00462 BC00462 V=166.7  +MOVJ EC00462
SMOVL C00463 BC00463 V=50.0 PL=0  +MOVJ EC00463
ARCON
SMOVL C00464 BC00464 V=9.2  +MOVJ EC00464
SMOVL C00465 BC00465 V=9.2  +MOVJ EC00465
ARCOF
SMOVL C00466 BC00466 V=1000.0  +MOVJ EC00466
SFTOF3D
'EndPath W4854
'12
MOVJ C00467 BC00467 VJ=100.00  +MOVJ EC00467 VJ=100.00
MOVJ C00468 BC00468 VJ=100.00  +MOVJ EC00468 VJ=100.00
MOVJ C00469 BC00469 VJ=100.00  +MOVJ EC00469 VJ=100.00
'Path W3485
SFTOF3D
SFTON3D P034
MOVJ C00470 BC00470 VJ=100.00  +MOVJ EC00470 VJ=100.00
SMOVL C00471 BC00471 V=800.0  +MOVJ EC00471
SMOVL C00472 BC00472 V=150.0 PL=0  +MOVJ EC00472
MACRO1 MJ#(0) ARGF14
ARCON
SMOVL C00473 BC00473 V=10.0  +MOVJ EC00473
SMOVL C00474 BC00474 V=10.0  +MOVJ EC00474
SMOVL C00475 BC00475 V=10.0  +MOVJ EC00475
ARCOF
SMOVL C00476 BC00476 V=800.0  +MOVJ EC00476
SMOVL C00477 BC00477 V=1000.0  +MOVJ EC00477
SFTOF3D
MOVJ C00478 BC00478 VJ=80.00  +MOVJ EC00478 VJ=80.00
MOVJ C00479 BC00479 VJ=80.00  +MOVJ EC00479 VJ=80.00
MOVJ C00480 BC00480 VJ=80.00  +MOVJ EC00480 VJ=80.00
MACRO1 MJ#(0) ARGF6
SFTON3D P063
SMOVL C00481 BC00481 V=166.7  +MOVJ EC00481
ARCON
SMOVL C00482 BC00482 V=11.7  +MOVJ EC00482
SMOVL C00483 BC00483 V=11.7  +MOVJ EC00483
SFTON3D P062
SMOVL C00484 BC00484 V=11.0  +MOVJ EC00484
SMOVL C00485 BC00485 V=11.0  +MOVJ EC00485
SFTON3D P061
SMOVL C00486 BC00486 V=11.0  +MOVJ EC00486
SMOVL C00487 BC00487 V=11.0  +MOVJ EC00487
ARCOF
SMOVL C00488 BC00488 V=800.0  +MOVJ EC00488
SFTOF3D
MOVJ C00489 BC00489 VJ=80.00  +MOVJ EC00489 VJ=80.00
MOVJ C00490 BC00490 VJ=80.00  +MOVJ EC00490 VJ=80.00
MOVJ C00491 BC00491 VJ=80.00  +MOVJ EC00491 VJ=80.00
'EndPath W3485
'Path W3486
SFTOF3D
SFTON3D P050
MOVJ C00492 BC00492 VJ=100.00  +MOVJ EC00492 VJ=100.00
SMOVL C00493 BC00493 V=800.0  +MOVJ EC00493
SMOVL C00494 BC00494 V=150.0 PL=0  +MOVJ EC00494
MACRO1 MJ#(0) ARGF14
ARCON
SMOVL C00495 BC00495 V=10.0  +MOVJ EC00495
SMOVL C00496 BC00496 V=10.0  +MOVJ EC00496
SMOVL C00497 BC00497 V=10.0  +MOVJ EC00497
ARCOF
SMOVL C00498 BC00498 V=800.0  +MOVJ EC00498
SMOVL C00499 BC00499 V=1000.0  +MOVJ EC00499
SFTOF3D
'EndPath W3486
MOVJ C00500 BC00500 VJ=100.00  +MOVJ EC00500 VJ=100.00
'Path W3485
SFTOF3D
SFTON3D P034
MOVJ C00501 BC00501 VJ=100.00  +MOVJ EC00501 VJ=100.00
SMOVL C00502 BC00502 V=800.0  +MOVJ EC00502
SMOVL C00503 BC00503 V=166.7 PL=0  +MOVJ EC00503
ARCON
SMOVL C00504 BC00504 V=9.2  +MOVJ EC00504
SMOVL C00505 BC00505 V=9.2  +MOVJ EC00505
SMOVL C00506 BC00506 V=9.2  +MOVJ EC00506
ARCOF
SMOVL C00507 BC00507 V=800.0  +MOVJ EC00507
SMOVL C00508 BC00508 V=1000.0  +MOVJ EC00508
SFTOF3D
'EndPath W3485
'Path W3487
SFTOF3D
SFTON3D P054
MOVJ C00509 BC00509 VJ=100.00  +MOVJ EC00509 VJ=100.00
SMOVL C00510 BC00510 V=800.0  +MOVJ EC00510
SMOVL C00511 BC00511 V=150.0 PL=0  +MOVJ EC00511
ARCON
SMOVL C00512 BC00512 V=9.2  +MOVJ EC00512
SMOVL C00513 BC00513 V=9.2  +MOVJ EC00513
SMOVL C00514 BC00514 V=9.2  +MOVJ EC00514
ARCOF
SMOVL C00515 BC00515 V=800.0  +MOVJ EC00515
SMOVL C00516 BC00516 V=1000.0  +MOVJ EC00516
SFTOF3D
'EndPath W3487
MOVJ C00517 BC00517 VJ=100.00  +MOVJ EC00517 VJ=100.00
'Path W3487
SFTOF3D
SFTON3D P028
MOVJ C00518 BC00518 VJ=100.00  +MOVJ EC00518 VJ=100.00
SMOVL C00519 BC00519 V=800.0  +MOVJ EC00519
SMOVL C00520 BC00520 V=150.0 PL=0  +MOVJ EC00520
ARCON
SMOVL C00521 BC00521 V=9.2  +MOVJ EC00521
SMOVL C00522 BC00522 V=9.2  +MOVJ EC00522
SMOVL C00523 BC00523 V=9.2  +MOVJ EC00523
ARCOF
SMOVL C00524 BC00524 V=800.0  +MOVJ EC00524
SMOVL C00525 BC00525 V=1000.0  +MOVJ EC00525
SFTOF3D
'EndPath W3487
MOVJ C00526 BC00526 VJ=100.00  +MOVJ EC00526 VJ=100.00
MOVJ C00527 BC00527 VJ=100.00  +MOVJ EC00527 VJ=100.00
'brak dostepu offset 5mm
'Path W3488
SFTOF3D
SFTON3D P028
MOVJ C00528 BC00528 VJ=100.00  +MOVJ EC00528 VJ=100.00
SMOVL C00529 BC00529 V=800.0  +MOVJ EC00529
SMOVL C00530 BC00530 V=150.0 PL=0  +MOVJ EC00530
ARCON
SMOVL C00531 BC00531 V=11.7  +MOVJ EC00531
ARCOF
SMOVL C00532 BC00532 V=800.0  +MOVJ EC00532
SMOVL C00533 BC00533 V=1000.0  +MOVJ EC00533
SFTOF3D
'EndPath W3488
MOVJ C00534 BC00534 VJ=100.00  +MOVJ EC00534 VJ=100.00
'13
'Path W3489
SFTOF3D
SFTON3D P030
MOVJ C00535 BC00535 VJ=100.00  +MOVJ EC00535 VJ=100.00
SMOVL C00536 BC00536 V=800.0  +MOVJ EC00536
SMOVL C00537 BC00537 V=150.0 PL=0  +MOVJ EC00537
MACRO1 MJ#(0) ARGF9
ARCON
SFTON3D P031
SMOVL C00538 BC00538 V=10.8  +MOVJ EC00538
ARCOF
SMOVL C00539 BC00539 V=800.0  +MOVJ EC00539
SMOVL C00540 BC00540 V=1000.0  +MOVJ EC00540
SFTOF3D
'EndPath W3489
'Path W3490
SFTOF3D
MOVJ C00541 BC00541 VJ=100.00  +MOVJ EC00541 VJ=100.00
MACRO1 MJ#(0) ARGF6
SFTON3D P069
SMOVL C00542 BC00542 V=250.0  +MOVJ EC00542
ARCON
SMOVL C00543 BC00543 V=11.7  +MOVJ EC00543
ARCOF
SMOVL C00544 BC00544 V=250.0  +MOVJ EC00544
SFTOF3D
SFTON3D P052
MOVJ C00545 BC00545 VJ=100.00  +MOVJ EC00545 VJ=100.00
SMOVL C00546 BC00546 V=800.0  +MOVJ EC00546
SMOVL C00547 BC00547 V=150.0 PL=0  +MOVJ EC00547
MACRO1 MJ#(0) ARGF14
ARCON
SMOVL C00548 BC00548 V=10.0  +MOVJ EC00548
SMOVL C00549 BC00549 V=10.0  +MOVJ EC00549
SMOVL C00550 BC00550 V=10.0  +MOVJ EC00550
ARCOF
SMOVL C00551 BC00551 V=800.0  +MOVJ EC00551
SMOVL C00552 BC00552 V=1000.0  +MOVJ EC00552
SFTOF3D
'EndPath W3490
MOVJ C00553 BC00553 VJ=100.00  +MOVJ EC00553 VJ=100.00
'poprawic spoine - nie mialem w
'yciecia
'Path W3491
SFTOF3D
SFTON3D P053
MOVJ C00554 BC00554 VJ=100.00  +MOVJ EC00554 VJ=100.00
SMOVL C00555 BC00555 V=800.0  +MOVJ EC00555
SMOVL C00556 BC00556 V=150.0 PL=0  +MOVJ EC00556
ARCON
SMOVL C00557 BC00557 V=10.0  +MOVJ EC00557
SMOVL C00558 BC00558 V=10.0  +MOVJ EC00558
SMOVL C00559 BC00559 V=10.0  +MOVJ EC00559
ARCOF
SMOVL C00560 BC00560 V=800.0  +MOVJ EC00560
SMOVL C00561 BC00561 V=1000.0  +MOVJ EC00561
SFTOF3D
'EndPath W3491
'14
'15-brak
MOVJ C00562 BC00562 VJ=100.00  +MOVJ EC00562 VJ=100.00
'16
'Path W3491
SFTOF3D
SFTON3D P029
MOVJ C00563 BC00563 VJ=100.00  +MOVJ EC00563 VJ=100.00
SMOVL C00564 BC00564 V=800.0  +MOVJ EC00564
SMOVL C00565 BC00565 V=150.0 PL=0  +MOVJ EC00565
ARCON
SMOVL C00566 BC00566 V=10.0  +MOVJ EC00566
SMOVL C00567 BC00567 V=10.0  +MOVJ EC00567
ARCOF
SMOVL C00568 BC00568 V=800.0  +MOVJ EC00568
SMOVL C00569 BC00569 V=1000.0  +MOVJ EC00569
SFTOF3D
'EndPath W3491
MOVJ C00570 BC00570 VJ=100.00  +MOVJ EC00570 VJ=100.00
'Path W3492
SFTOF3D
SFTON3D P029
MOVJ C00571 BC00571 VJ=100.00  +MOVJ EC00571 VJ=100.00
SMOVL C00572 BC00572 V=800.0  +MOVJ EC00572
SMOVL C00573 BC00573 V=150.0 PL=0  +MOVJ EC00573
ARCON
SMOVL C00574 BC00574 V=10.0  +MOVJ EC00574
ARCOF
SMOVL C00575 BC00575 V=800.0  +MOVJ EC00575
SMOVL C00576 BC00576 V=1000.0  +MOVJ EC00576
SFTOF3D
'EndPath W3492
MOVJ C00577 BC00577 VJ=100.00  +MOVJ EC00577 VJ=100.00
MOVJ C00578 BC00578 VJ=100.00  +MOVJ EC00578 VJ=100.00
'Path W3493
SFTOF3D
SFTON3D P029
MOVJ C00579 BC00579 VJ=100.00  +MOVJ EC00579 VJ=100.00
SMOVL C00580 BC00580 V=800.0  +MOVJ EC00580
SMOVL C00581 BC00581 V=150.0 PL=0  +MOVJ EC00581
ARCON
SMOVL C00582 BC00582 V=10.0  +MOVJ EC00582
SMOVL C00583 BC00583 V=10.0  +MOVJ EC00583
SMOVL C00584 BC00584 V=10.0  +MOVJ EC00584
ARCON
SMOVL C00585 BC00585 V=11.7  +MOVJ EC00585
ARCON
SMOVL C00586 BC00586 V=11.7  +MOVJ EC00586
ARCOF
SMOVL C00587 BC00587 V=800.0  +MOVJ EC00587
SMOVL C00588 BC00588 V=1000.0  +MOVJ EC00588
SFTOF3D
'EndPath W3493
MOVJ C00589 BC00589 VJ=100.00  +MOVJ EC00589 VJ=100.00
MOVJ C00590 BC00590 VJ=100.00  +MOVJ EC00590 VJ=100.00
'16
'Path W3491
SFTOF3D
SFTON3D P080
MOVJ C00591 BC00591 VJ=100.00  +MOVJ EC00591 VJ=100.00
SMOVL C00592 BC00592 V=800.0  +MOVJ EC00592
SMOVL C00593 BC00593 V=150.0 PL=0  +MOVJ EC00593
ARCON
SMOVL C00594 BC00594 V=10.0  +MOVJ EC00594
SMOVL C00595 BC00595 V=10.0  +MOVJ EC00595
ARCOF
SMOVL C00596 BC00596 V=800.0  +MOVJ EC00596
SMOVL C00597 BC00597 V=1000.0  +MOVJ EC00597
SFTOF3D
'EndPath W3491
MOVJ C00598 BC00598 VJ=100.00  +MOVJ EC00598 VJ=100.00
'Path W3492
SFTOF3D
SFTON3D P080
MOVJ C00599 BC00599 VJ=100.00  +MOVJ EC00599 VJ=100.00
SMOVL C00600 BC00600 V=800.0  +MOVJ EC00600
SMOVL C00601 BC00601 V=150.0 PL=0  +MOVJ EC00601
ARCON
SMOVL C00602 BC00602 V=10.0  +MOVJ EC00602
ARCOF
SMOVL C00603 BC00603 V=800.0  +MOVJ EC00603
SMOVL C00604 BC00604 V=1000.0  +MOVJ EC00604
SFTOF3D
'EndPath W3492
MOVJ C00605 BC00605 VJ=100.00  +MOVJ EC00605 VJ=100.00
MOVJ C00606 BC00606 VJ=100.00  +MOVJ EC00606 VJ=100.00
'Path W3493
SFTOF3D
SFTON3D P080
MOVJ C00607 BC00607 VJ=100.00  +MOVJ EC00607 VJ=100.00
SMOVL C00608 BC00608 V=800.0  +MOVJ EC00608
SMOVL C00609 BC00609 V=150.0 PL=0  +MOVJ EC00609
ARCON
SMOVL C00610 BC00610 V=10.0  +MOVJ EC00610
SMOVL C00611 BC00611 V=10.0  +MOVJ EC00611
SMOVL C00612 BC00612 V=10.0  +MOVJ EC00612
ARCON
SMOVL C00613 BC00613 V=11.7  +MOVJ EC00613
ARCON
SMOVL C00614 BC00614 V=11.7  +MOVJ EC00614
ARCOF
SMOVL C00615 BC00615 V=800.0  +MOVJ EC00615
SMOVL C00616 BC00616 V=1000.0  +MOVJ EC00616
SFTOF3D
'EndPath W3493
MOVJ C00617 BC00617 VJ=100.00  +MOVJ EC00617 VJ=100.00
MOVJ C00618 BC00618 VJ=100.00  +MOVJ EC00618 VJ=100.00
'17
'Path W3494
SFTOF3D
SFTON3D P027
MOVJ C00619 BC00619 VJ=100.00  +MOVJ EC00619 VJ=100.00
SMOVL C00620 BC00620 V=800.0  +MOVJ EC00620
SMOVL C00621 BC00621 V=150.0 PL=0  +MOVJ EC00621
ARCON
SMOVL C00622 BC00622 V=10.0  +MOVJ EC00622
ARCOF
SMOVL C00623 BC00623 V=800.0  +MOVJ EC00623
SMOVL C00624 BC00624 V=1000.0  +MOVJ EC00624
SFTOF3D
'EndPath W3494
'Path W3495
SFTOF3D
SFTON3D P027
MOVJ C00625 BC00625 VJ=100.00  +MOVJ EC00625 VJ=100.00
SMOVL C00626 BC00626 V=800.0  +MOVJ EC00626
SMOVL C00627 BC00627 V=150.0 PL=0  +MOVJ EC00627
ARCON
SMOVL C00628 BC00628 V=10.8  +MOVJ EC00628
ARCOF
SMOVL C00629 BC00629 V=800.0  +MOVJ EC00629
SMOVL C00630 BC00630 V=1000.0  +MOVJ EC00630
SFTOF3D
'EndPath W3495
'Path W3496
SFTOF3D
SFTON3D P027
MOVJ C00631 BC00631 VJ=100.00  +MOVJ EC00631 VJ=100.00
SFTOF3D
'EndPath W3496
MOVJ C00632 BC00632 VJ=100.00  +MOVJ EC00632 VJ=100.00
MOVJ C00633 BC00633 VJ=100.00  +MOVJ EC00633 VJ=100.00
MOVJ C00634 BC00634 VJ=100.00  +MOVJ EC00634 VJ=100.00
'18
'Path W3497
SFTOF3D
SFTON3D P024
MOVJ C00635 BC00635 VJ=100.00  +MOVJ EC00635 VJ=100.00
SMOVL C00636 BC00636 V=800.0  +MOVJ EC00636
SMOVL C00637 BC00637 V=150.0 PL=0  +MOVJ EC00637
ARCON
SMOVL C00638 BC00638 V=9.2  +MOVJ EC00638
SMOVL C00639 BC00639 V=9.2  +MOVJ EC00639
SMOVL C00640 BC00640 V=9.2  +MOVJ EC00640
SMOVL C00641 BC00641 V=9.2  +MOVJ EC00641
ARCOF
SMOVL C00642 BC00642 V=800.0  +MOVJ EC00642
SMOVL C00643 BC00643 V=1000.0  +MOVJ EC00643
SFTOF3D
'EndPath W3497
'
'Path W4855
SFTOF3D
SFTON3D P071
MOVJ C00644 BC00644 VJ=100.00  +MOVJ EC00644 VJ=100.00
SMOVL C00645 BC00645 V=800.0  +MOVJ EC00645
MACRO1 MJ#(0) ARGF9
SMOVL C00646 BC00646 V=150.0 PL=0  +MOVJ EC00646
ARCON
SMOVL C00647 BC00647 V=8.8  +MOVJ EC00647
SFTON3D P072
SMOVL C00648 BC00648 V=8.8  +MOVJ EC00648
SMOVL C00649 BC00649 V=8.8  +MOVJ EC00649
ARCOF
SMOVL C00650 BC00650 V=166.7  +MOVJ EC00650
SMOVL C00651 BC00651 V=800.0  +MOVJ EC00651
SMOVL C00652 BC00652 V=800.0  +MOVJ EC00652
SMOVL C00653 BC00653 V=800.0  +MOVJ EC00653
SFTON3D P072
SMOVL C00654 BC00654 V=166.7 PL=0  +MOVJ EC00654
ARCON
SMOVL C00655 BC00655 V=8.8  +MOVJ EC00655
SMOVL C00656 BC00656 V=8.8  +MOVJ EC00656
SMOVL C00657 BC00657 V=8.8  +MOVJ EC00657
SMOVL C00658 BC00658 V=8.8  +MOVJ EC00658
ARCOF
MOVL C00659 BC00659 V=166.7  +MOVJ EC00659 VJ=0.78
SMOVL C00660 BC00660 V=1000.0  +MOVJ EC00660
SFTOF3D
'EndPath W4855
'
'
MOVJ C00661 BC00661 VJ=100.00  +MOVJ EC00661 VJ=100.00
'19
MOVJ C00662 BC00662 VJ=100.00  +MOVJ EC00662 VJ=100.00
'Path W3499
SFTOF3D
SFTON3D P023
MOVJ C00663 BC00663 VJ=100.00  +MOVJ EC00663 VJ=100.00
SMOVL C00664 BC00664 V=800.0  +MOVJ EC00664
SMOVL C00665 BC00665 V=150.0 PL=0  +MOVJ EC00665
MACRO1 MJ#(0) ARGF6
ARCON
SWVON WEV#(66)
SMOVL C00666 BC00666 V=7.5  +MOVJ EC00666
SMOVL C00667 BC00667 V=7.5  +MOVJ EC00667
SMOVL C00668 BC00668 V=7.5  +MOVJ EC00668
ARCOF
SWVOF
SMOVL C00669 BC00669 V=800.0  +MOVJ EC00669
SMOVL C00670 BC00670 V=1000.0  +MOVJ EC00670
SFTOF3D
'EndPath W3499
MOVJ C00671 BC00671 VJ=100.00  +MOVJ EC00671 VJ=100.00
'Path W3500
SFTOF3D
SFTON3D P034
MOVJ C00672 BC00672 VJ=100.00  +MOVJ EC00672 VJ=100.00
SMOVL C00673 BC00673 V=800.0  +MOVJ EC00673
MACRO1 MJ#(0) ARGF9
SMOVL C00674 BC00674 V=150.0 PL=0  +MOVJ EC00674
ARCON
SMOVL C00675 BC00675 V=8.3  +MOVJ EC00675
SFTON3D P050
SMOVL C00676 BC00676 V=8.3  +MOVJ EC00676
SMOVL C00677 BC00677 V=8.3  +MOVJ EC00677
ARCOF
SMOVL C00678 BC00678 V=800.0  +MOVJ EC00678
SMOVL C00679 BC00679 V=1000.0  +MOVJ EC00679
SFTOF3D
'EndPath W3500
'Path W3501
SFTOF3D
SFTON3D P051
MOVJ C00680 BC00680 VJ=100.00  +MOVJ EC00680 VJ=100.00
SMOVL C00681 BC00681 V=800.0  +MOVJ EC00681
SMOVL C00682 BC00682 V=150.0 PL=0  +MOVJ EC00682
ARCON
SMOVL C00683 BC00683 V=7.5  +MOVJ EC00683
SMOVL C00684 BC00684 V=7.5  +MOVJ EC00684
SMOVL C00685 BC00685 V=7.5  +MOVJ EC00685
ARCOF
SMOVL C00686 BC00686 V=800.0  +MOVJ EC00686
SMOVL C00687 BC00687 V=1000.0  +MOVJ EC00687
SFTOF3D
'EndPath W3501
MOVJ C00688 BC00688 VJ=100.00  +MOVJ EC00688 VJ=100.00
'20
MOVJ C00689 BC00689 VJ=100.00  +MOVJ EC00689 VJ=100.00
MOVJ C00690 BC00690 VJ=100.00  +MOVJ EC00690 VJ=100.00
'offset 5mm
'Path W3500
SFTOF3D
SFTON3D P032
MOVJ C00691 BC00691 VJ=100.00  +MOVJ EC00691 VJ=100.00
SMOVL C00692 BC00692 V=800.0  +MOVJ EC00692
SMOVL C00693 BC00693 V=150.0 PL=0  +MOVJ EC00693
ARCON
SMOVL C00694 BC00694 V=9.2  +MOVJ EC00694
ARCOF
SMOVL C00695 BC00695 V=800.0  +MOVJ EC00695
SMOVL C00696 BC00696 V=1000.0  +MOVJ EC00696
SFTOF3D
'EndPath W3500
SFTOF3D
'EndPath W3502
'offset 5mm
'Path W3503
SFTOF3D
SFTON3D P032
MOVJ C00697 BC00697 VJ=100.00  +MOVJ EC00697 VJ=100.00
SMOVL C00698 BC00698 V=800.0  +MOVJ EC00698
SMOVL C00699 BC00699 V=150.0 PL=0  +MOVJ EC00699
ARCON
SMOVL C00700 BC00700 V=10.0  +MOVJ EC00700
ARCOF
SMOVL C00701 BC00701 V=800.0  +MOVJ EC00701
SMOVL C00702 BC00702 V=1000.0  +MOVJ EC00702
SFTOF3D
'EndPath W3503
MOVJ C00703 BC00703 VJ=100.00  +MOVJ EC00703 VJ=100.00
'Path W3504
SFTOF3D
SFTON3D P032
MOVJ C00704 BC00704 VJ=100.00  +MOVJ EC00704 VJ=100.00
SMOVL C00705 BC00705 V=800.0  +MOVJ EC00705
SMOVL C00706 BC00706 V=150.0 PL=0  +MOVJ EC00706
ARCON
SMOVL C00707 BC00707 V=11.7  +MOVJ EC00707
SMOVL C00708 BC00708 V=11.7  +MOVJ EC00708
ARCOF
SMOVL C00709 BC00709 V=800.0  +MOVJ EC00709
SMOVL C00710 BC00710 V=1000.0  +MOVJ EC00710
SFTOF3D
'EndPath W3504
MOVJ C00711 BC00711 VJ=100.00  +MOVJ EC00711 VJ=100.00
'21
MOVJ C00712 BC00712 VJ=100.00  +MOVJ EC00712 VJ=100.00
'Path W3505
SFTOF3D
SFTON3D P021
MOVJ C00713 BC00713 VJ=100.00  +MOVJ EC00713 VJ=100.00
SMOVL C00714 BC00714 V=800.0  +MOVJ EC00714
SMOVL C00715 BC00715 V=150.0 PL=0  +MOVJ EC00715
ARCON
SFTON3D P022
SMOVL C00716 BC00716 V=10.8  +MOVJ EC00716
SMOVL C00717 BC00717 V=11.7  +MOVJ EC00717
ARCOF
SMOVL C00718 BC00718 V=800.0  +MOVJ EC00718
SMOVL C00719 BC00719 V=1000.0  +MOVJ EC00719
SFTOF3D
'EndPath W3505
MOVJ C00720 BC00720 VJ=100.00  +MOVJ EC00720 VJ=100.00
'Path W3506
SFTOF3D
SFTON3D P095
MOVJ C00721 BC00721 VJ=100.00  +MOVJ EC00721 VJ=100.00
SMOVL C00722 BC00722 V=800.0  +MOVJ EC00722
SMOVL C00723 BC00723 V=150.0 PL=0  +MOVJ EC00723
MACRO1 MJ#(0) ARGF14
ARCON
SMOVL C00724 BC00724 V=10.0  +MOVJ EC00724
SMOVL C00725 BC00725 V=10.0  +MOVJ EC00725
SMOVL C00726 BC00726 V=10.0  +MOVJ EC00726
ARCOF
SMOVL C00727 BC00727 V=800.0  +MOVJ EC00727
SMOVL C00728 BC00728 V=1000.0  +MOVJ EC00728
SFTOF3D
'EndPath W3506
'Path W3507
SFTOF3D
SFTON3D P096
MOVJ C00729 BC00729 VJ=100.00  +MOVJ EC00729 VJ=100.00
SMOVL C00730 BC00730 V=800.0  +MOVJ EC00730
SMOVL C00731 BC00731 V=150.0 PL=0  +MOVJ EC00731
ARCON
SMOVL C00732 BC00732 V=10.0  +MOVJ EC00732
SMOVL C00733 BC00733 V=10.0  +MOVJ EC00733
ARCOF
SMOVL C00734 BC00734 V=800.0  +MOVJ EC00734
SMOVL C00735 BC00735 V=1000.0  +MOVJ EC00735
SFTOF3D
'EndPath W3507
MOVJ C00736 BC00736 VJ=100.00  +MOVJ EC00736 VJ=100.00
MOVJ C00737 BC00737 VJ=100.00  +MOVJ EC00737 VJ=100.00
'Path W4856
SFTOF3D
SFTON3D P071
MOVJ C00738 BC00738 VJ=100.00  +MOVJ EC00738 VJ=100.00
SMOVL C00739 BC00739 V=800.0  +MOVJ EC00739
SMOVL C00740 BC00740 V=150.0 PL=0  +MOVJ EC00740
ARCON
SMOVL C00741 BC00741 V=8.3  +MOVJ EC00741
SFTON3D P073
SMOVL C00742 BC00742 V=8.3  +MOVJ EC00742
SMOVL C00743 BC00743 V=8.3  +MOVJ EC00743
ARCOF
SMOVL C00744 BC00744 V=800.0  +MOVJ EC00744
SMOVL C00745 BC00745 V=1000.0  +MOVJ EC00745
SFTOF3D
'EndPath W4856
MOVJ C00746 BC00746 VJ=100.00  +MOVJ EC00746 VJ=100.00
MOVJ C00747 BC00747 VJ=50.00  +MOVJ EC00747 VJ=0.78
MOVJ C00748 BC00748 VJ=100.00  +MOVJ EC00748 VJ=50.00
SFTON3D P080
SMOVL C00749 BC00749 V=800.0  +MOVJ EC00749
SMOVL C00750 BC00750 V=150.0 PL=0  +MOVJ EC00750
ARCON
SMOVL C00751 BC00751 V=8.3  +MOVJ EC00751
SMOVL C00752 BC00752 V=8.3  +MOVJ EC00752
ARCOF
SMOVL C00753 BC00753 V=800.0  +MOVJ EC00753
SFTOF3D
SMOVL C00754 BC00754 V=1000.0  +MOVJ EC00754
MOVJ C00755 BC00755 VJ=100.00  +MOVJ EC00755 VJ=100.00
MOVJ C00756 BC00756 VJ=100.00  +MOVJ EC00756 VJ=100.00
MOVJ C00757 BC00757 VJ=100.00  +MOVJ EC00757 VJ=100.00
MOVJ C00758 BC00758 VJ=100.00  +MOVJ EC00758 VJ=100.00
SFTON3D P081
SMOVL C00759 BC00759 V=666.7  +MOVJ EC00759
SMOVL C00760 BC00760 V=166.7 PL=0  +MOVJ EC00760
ARCON
SMOVL C00761 BC00761 V=8.3  +MOVJ EC00761
SMOVL C00762 BC00762 V=8.3  +MOVJ EC00762
SMOVL C00763 BC00763 V=8.3  +MOVJ EC00763
ARCOF
SMOVL C00764 BC00764 V=333.3  +MOVJ EC00764
SFTOF3D
MOVL C00765 BC00765 V=1000.0  +MOVJ EC00765 VJ=100.00
MOVJ C00766 BC00766 VJ=100.00  +MOVJ EC00766 VJ=100.00
MOVJ C00767 BC00767 VJ=100.00  +MOVJ EC00767 VJ=100.00
'cut_wire_dol
'cut_wire_dol
'cut_wire_dol
CALL JOB:CLEAN-R1_KM_NEW
MOVJ C00768 BC00768 VJ=100.00  +MOVJ EC00768 VJ=100.00
MOVJ C00769 BC00769 VJ=100.00  +MOVJ EC00769 VJ=100.00
MOVJ C00770 BC00770 VJ=100.00  +MOVJ EC00770 VJ=100.00
'Path S4011
SFTOF3D
MOVJ C00771 BC00771 VJ=100.00  +MOVJ EC00771 VJ=100.00
MOVL C00772 BC00772 V=666.7  +MOVJ EC00772 VJ=100.00
SMOVL C00773 BC00773 V=166.7  +MOVJ EC00773
SREFP 3 C00774 BC00774  +REFP EC00774
CALL JOB:SEARCH-R1-S13D
SET P049 P006
SFTON3D P049
SMOVL C00775 BC00775 V=166.7  +MOVJ EC00775
SMOVL C00776 BC00776 V=166.7  +MOVJ EC00776
SREFP 3 C00777 BC00777  +REFP EC00777
CALL JOB:SEARCH-R1-S13D
SET P049 P006
SFTON3D P049
SMOVL C00778 BC00778 V=166.7  +MOVJ EC00778
MOVL C00779 BC00779 V=1000.0  +MOVJ EC00779 VJ=100.00
'EndPath S4011
'Path S4010
SFTOF3D
MOVJ C00780 BC00780 VJ=100.00  +MOVJ EC00780 VJ=100.00
SMOVL C00781 BC00781 V=666.7  +MOVJ EC00781
SMOVL C00782 BC00782 V=166.7  +MOVJ EC00782
SREFP 3 C00783 BC00783  +REFP EC00783
CALL JOB:SEARCH-R1-S13D
SET P048 P006
SFTON3D P048
SMOVL C00784 BC00784 V=166.7  +MOVJ EC00784
SMOVL C00785 BC00785 V=166.7  +MOVJ EC00785
SREFP 3 C00786 BC00786  +REFP EC00786
CALL JOB:SEARCH-R1-S13D
SET P048 P006
SFTON3D P048
SMOVL C00787 BC00787 V=233.3  +MOVJ EC00787
MOVL C00788 BC00788 V=1000.0  +MOVJ EC00788 VJ=100.00
'EndPath S4010
'Path S4009
SFTOF3D
MOVJ C00789 BC00789 VJ=100.00  +MOVJ EC00789 VJ=100.00
MOVL C00790 BC00790 V=666.7  +MOVJ EC00790 VJ=100.00
SMOVL C00791 BC00791 V=166.7  +MOVJ EC00791
SREFP 3 C00792 BC00792  +REFP EC00792
CALL JOB:SEARCH-R1-S13D
SET P047 P006
SFTON3D P047
SMOVL C00793 BC00793 V=166.7  +MOVJ EC00793
SMOVL C00794 BC00794 V=166.7  +MOVJ EC00794
SREFP 3 C00795 BC00795  +REFP EC00795
CALL JOB:SEARCH-R1-S13D
SET P047 P006
SFTON3D P047
SMOVL C00796 BC00796 V=166.7  +MOVJ EC00796
MOVL C00797 BC00797 V=1000.0  +MOVJ EC00797 VJ=100.00
'EndPath S4009
MOVJ C00798 BC00798 VJ=100.00  +MOVJ EC00798 VJ=100.00
'Path S4008
SFTOF3D
MOVJ C00799 BC00799 VJ=100.00  +MOVJ EC00799 VJ=100.00
MOVL C00800 BC00800 V=666.7  +MOVJ EC00800 VJ=100.00
SMOVL C00801 BC00801 V=166.7  +MOVJ EC00801
SREFP 3 C00802 BC00802  +REFP EC00802
CALL JOB:SEARCH-R1-S13D
SET P046 P006
SFTON3D P046
SMOVL C00803 BC00803 V=166.7  +MOVJ EC00803
SMOVL C00804 BC00804 V=166.7  +MOVJ EC00804
SREFP 3 C00805 BC00805  +REFP EC00805
CALL JOB:SEARCH-R1-S13D
SET P046 P006
SFTON3D P046
SMOVL C00806 BC00806 V=166.7  +MOVJ EC00806
MOVL C00807 BC00807 V=1000.0  +MOVJ EC00807 VJ=100.00
'EndPath S4008
'Path S4007
SFTOF3D
MOVJ C00808 BC00808 VJ=100.00  +MOVJ EC00808 VJ=100.00
MOVL C00809 BC00809 V=666.7  +MOVJ EC00809 VJ=100.00
SMOVL C00810 BC00810 V=166.7  +MOVJ EC00810
SREFP 3 C00811 BC00811  +REFP EC00811
CALL JOB:SEARCH-R1-S13D
SET P045 P006
SFTON3D P045
SMOVL C00812 BC00812 V=166.7  +MOVJ EC00812
SMOVL C00813 BC00813 V=166.7  +MOVJ EC00813
SMOVL C00814 BC00814 V=166.7  +MOVJ EC00814
SREFP 3 C00815 BC00815  +REFP EC00815
CALL JOB:SEARCH-R1-S13D
SET P045 P006
SFTON3D P045
SMOVL C00816 BC00816 V=166.7  +MOVJ EC00816
MOVL C00817 BC00817 V=1000.0  +MOVJ EC00817 VJ=100.00
'EndPath S4007
'Path S3506
SFTOF3D
MOVJ C00818 BC00818 VJ=100.00  +MOVJ EC00818 VJ=100.00
MOVL C00819 BC00819 V=666.7  +MOVJ EC00819 VJ=100.00
SMOVL C00820 BC00820 V=166.7  +MOVJ EC00820
SREFP 3 C00821 BC00821  +REFP EC00821
CALL JOB:SEARCH-R1-S13D
SET P044 P006
SFTON3D P044
SMOVL C00822 BC00822 V=166.7  +MOVJ EC00822
SMOVL C00823 BC00823 V=166.7  +MOVJ EC00823
SREFP 3 C00824 BC00824  +REFP EC00824
CALL JOB:SEARCH-R1-S13D
SET P044 P006
SFTON3D P044
SMOVL C00825 BC00825 V=166.7  +MOVJ EC00825
MOVL C00826 BC00826 V=1000.0  +MOVJ EC00826 VJ=100.00
'EndPath S3506
MOVJ C00827 BC00827 VJ=100.00  +MOVJ EC00827 VJ=100.00
MOVJ C00828 BC00828 VJ=100.00  +MOVJ EC00828 VJ=100.00
MOVJ C00829 BC00829 VJ=100.00  +MOVJ EC00829 VJ=100.00
MOVJ C00830 BC00830 VJ=100.00  +MOVJ EC00830 VJ=100.00
MOVJ C00831 BC00831 VJ=100.00  +MOVJ EC00831 VJ=100.00
'Path S4006
SFTOF3D
MOVJ C00832 BC00832 VJ=100.00  +MOVJ EC00832 VJ=100.00
MOVL C00833 BC00833 V=666.7  +MOVJ EC00833 VJ=100.00
SMOVL C00834 BC00834 V=166.7  +MOVJ EC00834
SREFP 3 C00835 BC00835  +REFP EC00835
CALL JOB:SEARCH-R1-S13D
SET P043 P006
SFTON3D P043
SMOVL C00836 BC00836 V=166.7  +MOVJ EC00836
SMOVL C00837 BC00837 V=166.7  +MOVJ EC00837
SMOVL C00838 BC00838 V=166.7  +MOVJ EC00838
SREFP 3 C00839 BC00839  +REFP EC00839
CALL JOB:SEARCH-R1-S13D
SET P043 P006
SFTON3D P043
SMOVL C00840 BC00840 V=166.7  +MOVJ EC00840
MOVL C00841 BC00841 V=1000.0  +MOVJ EC00841 VJ=100.00
'EndPath S4006
'Path S4005
SFTOF3D
MOVJ C00842 BC00842 VJ=100.00  +MOVJ EC00842 VJ=100.00
MOVL C00843 BC00843 V=800.0  +MOVJ EC00843 VJ=100.00
SMOVL C00844 BC00844 V=166.7  +MOVJ EC00844
SREFP 3 C00845 BC00845  +REFP EC00845
CALL JOB:SEARCH-R1-S13D
SET P042 P006
SFTON3D P042
SMOVL C00846 BC00846 V=166.7  +MOVJ EC00846
SMOVL C00847 BC00847 V=166.7  +MOVJ EC00847
SREFP 3 C00848 BC00848  +REFP EC00848
CALL JOB:SEARCH-R1-S13D
SET P042 P006
SFTON3D P042
SMOVL C00849 BC00849 V=166.7  +MOVJ EC00849
MOVL C00850 BC00850 V=1000.0  +MOVJ EC00850 VJ=100.00
'EndPath S4005
'Path S4004
SFTOF3D
MOVJ C00851 BC00851 VJ=100.00  +MOVJ EC00851 VJ=100.00
MOVL C00852 BC00852 V=800.0  +MOVJ EC00852 VJ=100.00
SMOVL C00853 BC00853 V=166.7  +MOVJ EC00853
SMOVL C00854 BC00854 V=166.7  +MOVJ EC00854
SREFP 3 C00855 BC00855  +REFP EC00855
CALL JOB:SEARCH-R1-S13D
SET P041 P006
SFTON3D P041
SMOVL C00856 BC00856 V=166.7  +MOVJ EC00856
SMOVL C00857 BC00857 V=166.7  +MOVJ EC00857
SREFP 3 C00858 BC00858  +REFP EC00858
CALL JOB:SEARCH-R1-S13D
SET P041 P006
SFTON3D P041
SMOVL C00859 BC00859 V=166.7  +MOVJ EC00859
SREFP 3 C00860 BC00860  +REFP EC00860
CALL JOB:SEARCH-R1-S13D
SET P041 P006
SFTON3D P041
SMOVL C00861 BC00861 V=166.7  +MOVJ EC00861
MOVL C00862 BC00862 V=1000.0  +MOVJ EC00862 VJ=100.00
'EndPath S4004
'Path S4003
SFTOF3D
MOVJ C00863 BC00863 VJ=100.00  +MOVJ EC00863 VJ=100.00
MOVL C00864 BC00864 V=800.0  +MOVJ EC00864 VJ=100.00
SMOVL C00865 BC00865 V=166.7  +MOVJ EC00865
SREFP 3 C00866 BC00866  +REFP EC00866
CALL JOB:SEARCH-R1-S13D
SET P040 P006
SFTON3D P040
SMOVL C00867 BC00867 V=250.0  +MOVJ EC00867
SMOVL C00868 BC00868 V=250.0  +MOVJ EC00868
SMOVL C00869 BC00869 V=166.7  +MOVJ EC00869
SREFP 3 C00870 BC00870  +REFP EC00870
CALL JOB:SEARCH-R1-S13D
SET P040 P006
SFTON3D P040
SMOVL C00871 BC00871 V=166.7  +MOVJ EC00871
SMOVL C00872 BC00872 V=166.7  +MOVJ EC00872
SREFP 3 C00873 BC00873  +REFP EC00873
CALL JOB:SEARCH-R1-S13D
SET P040 P006
SFTON3D P040
SMOVL C00874 BC00874 V=166.7  +MOVJ EC00874
MOVL C00875 BC00875 V=1000.0  +MOVJ EC00875 VJ=100.00
'EndPath S4003
'Path W4012
SFTOF3D
SFTON3D P040
MOVJ C00876 BC00876 VJ=100.00  +MOVJ EC00876 VJ=100.00
SMOVL C00877 BC00877 V=800.0  +MOVJ EC00877
SMOVL C00878 BC00878 V=150.0 PL=0  +MOVJ EC00878
ARCON
SMOVL C00879 BC00879 V=11.7  +MOVJ EC00879
ARCOF
SMOVL C00880 BC00880 V=800.0  +MOVJ EC00880
SMOVL C00881 BC00881 V=1000.0  +MOVJ EC00881
SFTOF3D
'EndPath W4012
'Path W4013
SFTOF3D
SFTON3D P040
MOVJ C00882 BC00882 VJ=100.00  +MOVJ EC00882 VJ=100.00
SMOVL C00883 BC00883 V=800.0  +MOVJ EC00883
SMOVL C00884 BC00884 V=150.0 PL=0  +MOVJ EC00884
ARCON
SMOVL C00885 BC00885 V=10.0  +MOVJ EC00885
ARCOF
SMOVL C00886 BC00886 V=800.0  +MOVJ EC00886
SMOVL C00887 BC00887 V=1000.0  +MOVJ EC00887
SMOVL C00888 BC00888 V=1000.0  +MOVJ EC00888
SFTOF3D
'EndPath W4013
'Path W4014
SFTOF3D
SFTON3D P040
MOVJ C00889 BC00889 VJ=100.00  +MOVJ EC00889 VJ=100.00
SMOVL C00890 BC00890 V=800.0  +MOVJ EC00890
SMOVL C00891 BC00891 V=150.0 PL=0  +MOVJ EC00891
ARCON
SMOVL C00892 BC00892 V=10.0  +MOVJ EC00892
ARCOF
SMOVL C00893 BC00893 V=800.0  +MOVJ EC00893
SMOVL C00894 BC00894 V=1000.0  +MOVJ EC00894
SFTOF3D
'EndPath W4014
'
MOVJ C00895 BC00895 VJ=100.00  +MOVJ EC00895 VJ=100.00
MOVJ C00896 BC00896 VJ=100.00  +MOVJ EC00896 VJ=100.00
MOVJ C00897 BC00897 VJ=100.00  +MOVJ EC00897 VJ=100.00
MOVJ C00898 BC00898 VJ=100.00  +MOVJ EC00898 VJ=100.00
MOVJ C00899 BC00899 VJ=100.00  +MOVJ EC00899 VJ=100.00
'Path W3522
SFTOF3D
SFTON3D P045
MOVJ C00900 BC00900 VJ=100.00  +MOVJ EC00900 VJ=100.00
SMOVL C00901 BC00901 V=800.0  +MOVJ EC00901
SMOVL C00902 BC00902 V=150.0 PL=0  +MOVJ EC00902
MACRO1 MJ#(0) ARGF9
ARCON
SMOVL C00903 BC00903 V=11.7  +MOVJ EC00903
ARCOF
SMOVL C00904 BC00904 V=800.0  +MOVJ EC00904
SMOVL C00905 BC00905 V=1000.0  +MOVJ EC00905
SFTOF3D
'EndPath W3522
'Path W3520
SFTOF3D
SFTON3D P044
MOVJ C00906 BC00906 VJ=100.00  +MOVJ EC00906 VJ=100.00
SMOVL C00907 BC00907 V=800.0  +MOVJ EC00907
SMOVL C00908 BC00908 V=166.7 PL=0  +MOVJ EC00908
ARCON
SMOVL C00909 BC00909 V=11.7  +MOVJ EC00909
SMOVL C00910 BC00910 V=11.7  +MOVJ EC00910
SMOVL C00911 BC00911 V=11.7  +MOVJ EC00911
ARCOF
SMOVL C00912 BC00912 V=800.0  +MOVJ EC00912
SMOVL C00913 BC00913 V=1000.0  +MOVJ EC00913
SFTOF3D
'EndPath W3520
'Path W3519
SFTOF3D
SFTON3D P046
MOVJ C00914 BC00914 VJ=100.00  +MOVJ EC00914 VJ=100.00
SMOVL C00915 BC00915 V=800.0  +MOVJ EC00915
SMOVL C00916 BC00916 V=166.7 PL=0  +MOVJ EC00916
ARCON
SMOVL C00917 BC00917 V=12.5  +MOVJ EC00917
SMOVL C00918 BC00918 V=12.5  +MOVJ EC00918
SMOVL C00919 BC00919 V=12.5  +MOVJ EC00919
ARCOF
SMOVL C00920 BC00920 V=800.0  +MOVJ EC00920
SMOVL C00921 BC00921 V=1000.0  +MOVJ EC00921
SFTOF3D
'EndPath W3519
'1
MOVJ C00922 BC00922 VJ=100.00  +MOVJ EC00922 VJ=100.00
MOVJ C00923 BC00923 VJ=100.00  +MOVJ EC00923 VJ=100.00
'Path W3509
SFTOF3D
SFTON3D P048
MOVJ C00924 BC00924 VJ=100.00  +MOVJ EC00924 VJ=100.00
SMOVL C00925 BC00925 V=800.0  +MOVJ EC00925
SMOVL C00926 BC00926 V=150.0 PL=0  +MOVJ EC00926
ARCON
SMOVL C00927 BC00927 V=11.7  +MOVJ EC00927
ARCOF
SMOVL C00928 BC00928 V=800.0  +MOVJ EC00928
SMOVL C00929 BC00929 V=1000.0  +MOVJ EC00929
SFTOF3D
'EndPath W3509
'Path W3510
SFTOF3D
SFTON3D P049
MOVJ C00930 BC00930 VJ=100.00  +MOVJ EC00930 VJ=100.00
SMOVL C00931 BC00931 V=800.0  +MOVJ EC00931
SMOVL C00932 BC00932 V=150.0 PL=0  +MOVJ EC00932
MACRO1 MJ#(0) ARGF6
ARCON
SMOVL C00933 BC00933 V=9.2  +MOVJ EC00933
SMOVL C00934 BC00934 V=9.2  +MOVJ EC00934
SMOVL C00935 BC00935 V=9.2  +MOVJ EC00935
SMOVL C00936 BC00936 V=9.2  +MOVJ EC00936
SMOVL C00937 BC00937 V=9.2  +MOVJ EC00937
ARCOF
MOVJ C00938 BC00938 VJ=30.00  +MOVJ EC00938 VJ=80.00
MOVJ C00939 BC00939 VJ=30.00  +MOVJ EC00939 VJ=30.00
SMOVL C00940 BC00940 V=166.7  +MOVJ EC00940
ARCON
SMOVL C00941 BC00941 V=13.3  +MOVJ EC00941
SMOVL C00942 BC00942 V=13.3  +MOVJ EC00942
SMOVL C00943 BC00943 V=13.3  +MOVJ EC00943
ARCOF
SMOVL C00944 BC00944 V=333.3  +MOVJ EC00944
SMOVL C00945 BC00945 V=666.7  +MOVJ EC00945
SMOVL C00946 BC00946 V=166.7  +MOVJ EC00946
ARCON
SMOVL C00947 BC00947 V=13.3  +MOVJ EC00947
SMOVL C00948 BC00948 V=13.3  +MOVJ EC00948
ARCOF
SMOVL C00949 BC00949 V=166.7  +MOVJ EC00949
ARCON
SMOVL C00950 BC00950 V=11.7  +MOVJ EC00950
ARCOF
SMOVL C00951 BC00951 V=250.0  +MOVJ EC00951
SFTOF3D
'EndPath W3510
MOVJ C00952 BC00952 VJ=100.00  +MOVJ EC00952 VJ=100.00
'2
MOVJ C00953 BC00953 VJ=100.00  +MOVJ EC00953 VJ=100.00
MOVJ C00954 BC00954 VJ=100.00  +MOVJ EC00954 VJ=100.00
MOVJ C00955 BC00955 VJ=100.00  +MOVJ EC00955 VJ=100.00
'Path W3511
SFTOF3D
SFTON3D P043
MOVJ C00956 BC00956 VJ=100.00  +MOVJ EC00956 VJ=100.00
SMOVL C00957 BC00957 V=800.0  +MOVJ EC00957
SMOVL C00958 BC00958 V=166.7 PL=0  +MOVJ EC00958
MACRO1 MJ#(0) ARGF9
ARCON
SMOVL C00959 BC00959 V=11.7  +MOVJ EC00959
ARCOF
SMOVL C00960 BC00960 V=800.0  +MOVJ EC00960
SMOVL C00961 BC00961 V=1000.0  +MOVJ EC00961
SFTOF3D
'EndPath W3511
'Path W3512
SFTOF3D
SFTON3D P042
MOVJ C00962 BC00962 VJ=100.00  +MOVJ EC00962 VJ=100.00
SMOVL C00963 BC00963 V=800.0  +MOVJ EC00963
SMOVL C00964 BC00964 V=150.0 PL=0  +MOVJ EC00964
ARCON
SMOVL C00965 BC00965 V=11.7  +MOVJ EC00965
ARCOF
SMOVL C00966 BC00966 V=800.0  +MOVJ EC00966
SMOVL C00967 BC00967 V=1000.0  +MOVJ EC00967
SFTOF3D
'EndPath W3512
'3
MOVJ C00968 BC00968 VJ=100.00  +MOVJ EC00968 VJ=100.00
MOVJ C00969 BC00969 VJ=100.00  +MOVJ EC00969 VJ=100.00
MOVJ C00970 BC00970 VJ=100.00  +MOVJ EC00970 VJ=100.00
MOVJ C00971 BC00971 VJ=100.00  +MOVJ EC00971 VJ=100.00
'Path W3514
SFTOF3D
SFTON3D P047
MOVJ C00972 BC00972 VJ=100.00  +MOVJ EC00972 VJ=100.00
SMOVL C00973 BC00973 V=800.0  +MOVJ EC00973
SMOVL C00974 BC00974 V=150.0 PL=0  +MOVJ EC00974
ARCON
SMOVL C00975 BC00975 V=11.7  +MOVJ EC00975
ARCOF
SMOVL C00976 BC00976 V=800.0  +MOVJ EC00976
SMOVL C00977 BC00977 V=1000.0  +MOVJ EC00977
SFTOF3D
'EndPath W3514
'Path W3518
SFTOF3D
SFTON3D P047
MOVJ C00978 BC00978 VJ=100.00  +MOVJ EC00978 VJ=100.00
SMOVL C00979 BC00979 V=800.0  +MOVJ EC00979
SMOVL C00980 BC00980 V=150.0 PL=0  +MOVJ EC00980
ARCON
SMOVL C00981 BC00981 V=11.7  +MOVJ EC00981
ARCOF
SMOVL C00982 BC00982 V=800.0  +MOVJ EC00982
SMOVL C00983 BC00983 V=1000.0  +MOVJ EC00983
SFTOF3D
'EndPath W3518
MOVJ C00984 BC00984 VJ=100.00  +MOVJ EC00984 VJ=100.00
MOVJ C00985 BC00985 VJ=100.00  +MOVJ EC00985 VJ=100.00
MOVJ C00986 BC00986 VJ=100.00  +MOVJ EC00986 VJ=100.00
MOVJ C00987 BC00987 VJ=100.00  +MOVJ EC00987 VJ=100.00
'Path W3516
SFTOF3D
SFTON3D P043
MOVJ C00988 BC00988 VJ=50.00  +MOVJ EC00988 VJ=50.00
MOVJ C00989 BC00989 VJ=100.00  +MOVJ EC00989 VJ=100.00
SMOVL C00990 BC00990 V=800.0  +MOVJ EC00990
SMOVL C00991 BC00991 V=150.0 PL=0  +MOVJ EC00991
ARCON
SMOVL C00992 BC00992 V=11.7  +MOVJ EC00992
ARCOF
SMOVL C00993 BC00993 V=800.0  +MOVJ EC00993
SMOVL C00994 BC00994 V=1000.0  +MOVJ EC00994
SFTOF3D
'EndPath W3516
'Path W3515
SFTOF3D
SFTON3D P042
MOVJ C00995 BC00995 VJ=100.00  +MOVJ EC00995 VJ=100.00
SMOVL C00996 BC00996 V=800.0  +MOVJ EC00996
SMOVL C00997 BC00997 V=166.7 PL=0  +MOVJ EC00997
ARCON
SMOVL C00998 BC00998 V=10.8  +MOVJ EC00998
ARCOF
SMOVL C00999 BC00999 V=800.0  +MOVJ EC00999
SMOVL C01000 BC01000 V=1000.0  +MOVJ EC01000
SFTOF3D
'EndPath W3515
MOVJ C01001 BC01001 VJ=100.00  +MOVJ EC01001 VJ=100.00
MOVJ C01002 BC01002 VJ=100.00  +MOVJ EC01002 VJ=100.00
MOVJ C01003 BC01003 VJ=100.00  +MOVJ EC01003 VJ=100.00
MOVJ C01004 BC01004 VJ=100.00  +MOVJ EC01004 VJ=100.00
'Path W3523
SFTOF3D
SFTON3D P046
MOVJ C01005 BC01005 VJ=100.00  +MOVJ EC01005 VJ=100.00
SMOVL C01006 BC01006 V=800.0  +MOVJ EC01006
SMOVL C01007 BC01007 V=166.7 PL=0  +MOVJ EC01007
MACRO1 MJ#(0) ARGF14
ARCON
SMOVL C01008 BC01008 V=10.0  +MOVJ EC01008
ARCOF
SMOVL C01009 BC01009 V=800.0  +MOVJ EC01009
SMOVL C01010 BC01010 V=1000.0  +MOVJ EC01010
SFTOF3D
'EndPath W3523
'Path W4015
SFTOF3D
SFTON3D P044
MOVJ C01011 BC01011 VJ=100.00  +MOVJ EC01011 VJ=100.00
SMOVL C01012 BC01012 V=800.0  +MOVJ EC01012
SMOVL C01013 BC01013 V=150.0 PL=0  +MOVJ EC01013
MACRO1 MJ#(0) ARGF9
ARCON
SMOVL C01014 BC01014 V=10.8  +MOVJ EC01014
ARCOF
SMOVL C01015 BC01015 V=800.0  +MOVJ EC01015
SMOVL C01016 BC01016 V=1000.0  +MOVJ EC01016
SFTOF3D
'EndPath W4015
MOVJ C01017 BC01017 VJ=100.00  +MOVJ EC01017 VJ=100.00
MOVJ C01018 BC01018 VJ=100.00  +MOVJ EC01018 VJ=100.00
MOVJ C01019 BC01019 VJ=100.00  +MOVJ EC01019 VJ=100.00
MOVJ C01020 BC01020 VJ=100.00  +MOVJ EC01020 VJ=100.00
'Path W4016
SFTOF3D
SFTON3D P041
MOVJ C01021 BC01021 VJ=100.00  +MOVJ EC01021 VJ=100.00
SMOVL C01022 BC01022 V=800.0  +MOVJ EC01022
SMOVL C01023 BC01023 V=150.0 PL=0  +MOVJ EC01023
MACRO1 MJ#(0) ARGF14
ARCON
SMOVL C01024 BC01024 V=10.0  +MOVJ EC01024
SMOVL C01025 BC01025 V=10.0  +MOVJ EC01025
SMOVL C01026 BC01026 V=10.0  +MOVJ EC01026
ARCOF
SMOVL C01027 BC01027 V=800.0  +MOVJ EC01027
SMOVL C01028 BC01028 V=1000.0  +MOVJ EC01028
SFTOF3D
'EndPath W4016
'Path W4017
SFTOF3D
SFTON3D P041
MOVJ C01029 BC01029 VJ=100.00  +MOVJ EC01029 VJ=100.00
SMOVL C01030 BC01030 V=800.0  +MOVJ EC01030
SMOVL C01031 BC01031 V=150.0 PL=0  +MOVJ EC01031
SMOVL C01032 BC01032 V=10.0  +MOVJ EC01032
ARCOF
SMOVL C01033 BC01033 V=800.0  +MOVJ EC01033
SMOVL C01034 BC01034 V=1000.0  +MOVJ EC01034
SFTOF3D
'EndPath W4017
MOVJ C01035 BC01035 VJ=100.00  +MOVJ EC01035 VJ=100.00
'Path W4018
SFTOF3D
SFTON3D P041
MOVJ C01036 BC01036 VJ=100.00  +MOVJ EC01036 VJ=100.00
SMOVL C01037 BC01037 V=800.0  +MOVJ EC01037
SMOVL C01038 BC01038 V=150.0 PL=0  +MOVJ EC01038
SMOVL C01039 BC01039 V=10.0  +MOVJ EC01039
ARCOF
SMOVL C01040 BC01040 V=800.0  +MOVJ EC01040
SMOVL C01041 BC01041 V=1000.0  +MOVJ EC01041
SFTOF3D
'EndPath W4018
MOVJ C01042 BC01042 VJ=100.00  +MOVJ EC01042 VJ=100.00
MOVJ C01043 BC01043 VJ=100.00  +MOVJ EC01043 VJ=100.00
MOVJ C01044 BC01044 VJ=100.00  +MOVJ EC01044 VJ=100.00
MOVJ C01045 BC01045 VJ=100.00  +MOVJ EC01045 VJ=100.00
MOVJ C01046 BC01046 VJ=100.00  +MOVJ EC01046 VJ=100.00
END
